# B&R Automation Studio project Panasonic_LinkaPowerCP2_A2021055 (part 40)

#### Main.st - Init, cyclic, exit code
```iecst
PROGRAM _INIT
	(* Insert code here *)

END_PROGRAM

PROGRAM _CYCLIC

	//Volanie funkcie SequenceControl//
    SequenceControl(SC:= SC_Devlink);

    //******************************************Štruktura nazvu adresára na serveri Panasonic************************************************//
    //Názov linky//
    StruktNovehoNazvuAdresara.LINKA:= 'PowerCP_CP4';

    //Názov pracoviska//
    StruktNovehoNazvuAdresara.PRACOVISKO:= 'ST10';

    //Rok//
    brsstrcpy(ADR(StruktNovehoNazvuAdresara.ROK),ADR(Rok_STR_4_Znaky));

    //Dátum//
    StruktNovehoNazvuAdresara.DATUM:= '';
    brsstrcat(ADR(StruktNovehoNazvuAdresara.DATUM),ADR(Rok_STR_4_Znaky));
    brsstrcat(ADR(StruktNovehoNazvuAdresara.DATUM),ADR('_'));
    brsstrcat(ADR(StruktNovehoNazvuAdresara.DATUM),ADR(Mesiac_STR));
    brsstrcat(ADR(StruktNovehoNazvuAdresara.DATUM),ADR('_'));
    brsstrcat(ADR(StruktNovehoNazvuAdresara.DATUM),ADR(Den_STR));

    //*********************************************Štruktura názvu premenovaného súboru v PLC***************************************************//
    //Datum//
    StruktNovehoNazvuSuboru.DATUM:= '';
    brsstrcat(ADR(StruktNovehoNazvuSuboru.DATUM),ADR(Rok_STR_4_Znaky));
    brsstrcat(ADR(StruktNovehoNazvuSuboru.DATUM),ADR('_'));
    brsstrcat(ADR(StruktNovehoNazvuSuboru.DATUM),ADR(Mesiac_STR));
    brsstrcat(ADR(StruktNovehoNazvuSuboru.DATUM),ADR('_'));
    brsstrcat(ADR(StruktNovehoNazvuSuboru.DATUM),ADR(Den_STR));

    //Čas//
    StruktNovehoNazvuSuboru.CAS:= '';
    brsstrcat(ADR(StruktNovehoNazvuSuboru.CAS),ADR(Hodina_STR));
    brsstrcat(ADR(StruktNovehoNazvuSuboru.CAS),ADR('_'));
    brsstrcat(ADR(StruktNovehoNazvuSuboru.CAS),ADR(Minuta_STR));
    brsstrcat(ADR(StruktNovehoNazvuSuboru.CAS),ADR('_'));
    brsstrcat(ADR(StruktNovehoNazvuSuboru.CAS),ADR(Sekunda_STR));

    //Kód modelu//
    StruktNovehoNazvuSuboru.SERIAL:= FTP_CAM16.INPUTS.QRkodPowerCP;

    //Index fotky//
    StruktNovehoNazvuSuboru.INDEX:= FTP_CAM16.INPUTS.IndexFotky;

    //Result fotky//
    StruktNovehoNazvuSuboru.RESULT:= FTP_CAM16.INPUTS.Result;

	//Prípona súboru//
	IF TypFotky_BMP THEN
		StruktNovehoNazvuSuboru.Pripona:= '.bmp';
	ELSE
		StruktNovehoNazvuSuboru.Pripona:= '.jpg';
	END_IF

    //Mapovanie premenných//
    FTP_CAM16.STATUS.AdresarPrazdny:= AdresarPrazdny;

	CASE SC_Devlink.Step OF

		0:
			SC_Devlink.StepName:= '0 - Nulovanie';
			FTP_CAM16.STATUS.KomunikaciaError:= FALSE;
			FTP_CAM16.STATUS.KomunikaciaUkoncena:= FALSE;
			PocetHladaniFotky:= 0;
            AdresarPrazdny:= FALSE;
            PocetNajdenychSuborov:= 0;
            PocetNajdenychAdresarov:= 0;
            PocetPremenovanychSuborov:= 0;
            PocetSkopirovanychSuborov:= 0;
            PocetVymazanychSuborov:= 0;
            i:= 0;
            PocetPokusov_FTP_KOM:= 0;
			PoruchaKomunikacie:= FALSE;
			DirInfo_0.enable:= FALSE;
			DirRead_0.enable:= FALSE;
			FileRename_0.enable:= FALSE;
			DirCreate_0.enable:= FALSE;
			DirInfo_0.enable:= FALSE;
			DirRead_0.enable:= FALSE;
			FileCopy_0.enable:= FALSE;
			FileDelete_0.enable:= FALSE;
			SC_Devlink.Step:= 1;

        1:
            SC_Devlink.StepName:= '1 - Rozhodnutie o cinnosti';
            IF FTP_CAM16.CMD.OdosliFotku THEN
                FTP_CAM16.STATUS.PopisPoruchy:= '';
                SC_Devlink.Step:= 15;
            ELSIF FTP_CAM16.CMD.VymazFotku THEN
                FTP_CAM16.STATUS.PopisPoruchy:= '';
                SC_Devlink.Step:= 153;
            END_IF

		15:
			SC_Devlink.StepName:= '15 - Odoslanie fotky, kontrola pripojenia na FTP server Panasonic';
			SC_Devlink.IdleTime.PT:= T#3s;
			SC_Devlink.AlarmTime.PT:= T#3s;

			IF Stav_PripojenieFTP_OK THEN
				SC_Devlink.ResetStep:= TRUE;
				SC_Devlink.Step:= 20;
			END_IF

        20:
            SC_Devlink.StepName:= '20 - Odoslanie fotky na server, nacitanie adresara kamery pred premenovanim';
            SC_Devlink.IdleTime.PT:= T#3s;
            SC_Devlink.AlarmTime.PT:= T#3s;

            DirInfo_0.enable:= TRUE;
            DirInfo_0.pDevice:= ADR('CAM16');
            DirInfo_0.pPath:= ADR('/');   //ak je nula tak číta všetky súbory a adresáre v koreni ak je "/Temp" tak číta všetky súbory a adresáre v adresári Temp//
            DirInfo_0();

            IF DirInfo_0.status = 0 THEN
                PocetNajdenychAdresarov:= DirInfo_0.dirnum;
                PocetNajdenychSuborov:= DirInfo_0.filenum;
                brsmemset(ADR(FileList[0]),0, SIZEOF(FileList));  //Vynulovanie pola stringov pre záznam adresárov a súborov
                SC_Devlink.ResetStep:= TRUE;
                SC_Devlink.Step:= 23;
            ELSIF DirInfo_0.status = 65535 THEN
                //BUSY//
            ELSIF DirInfo_0.status = 20723 THEN
                FTP_CAM16.STATUS.PopisPoruchy:= 'Porucha nacitania adresara kamery';
                Buffer_16.Hodnota:= DirInfo_0.status;
                Buffer_16.ZapisHodnotu:= TRUE;
                PoruchaKomunikacie:= TRUE;
                SC_Devlink.ResetStep:= TRUE;
                SC_Devlink.Step:= 100;
            ELSE
                FTP_CAM16.STATUS.PopisPoruchy:= 'Porucha nacitania adresara kamery';
                IF DirInfo_0.status = 20799 THEN
                    Buffer_16.Hodnota:= FileIoGetSysError();
                ELSE
                    Buffer_16.Hodnota:= DirInfo_0.status;
                END_IF
                Buffer_16.ZapisHodnotu:= TRUE;
                PoruchaKomunikacie:= TRUE;
                SC_Devlink.ResetStep:= TRUE;
                SC_Devlink.Step:= 100;
            END_IF

        23:
            SC_Devlink.StepName:= '23 - Odoslanie fotky na server, kontrola poctu najdenych suborov v adresari kamery';
            SC_Devlink.IdleTime.PT:= T#3s;
            SC_Devlink.AlarmTime.PT:= T#3s;

            IF PocetNajdenychSuborov > 0 THEN
                PocetHladaniFotky:= 0;
                SC_Devlink.ResetStep:= TRUE;
                SC_Devlink.Step:= 25;
            ELSIF PocetHladaniFotky < 100 THEN
                PocetHladaniFotky:= PocetHladaniFotky + 1;
                SC_Devlink.ResetStep:= TRUE;
                SC_Devlink.Step:= 20;
            ELSIF PocetHladaniFotky >= 100 THEN
                AdresarPrazdny:= TRUE;
                FTP_CAM16.STATUS.KomunikaciaUkoncena:= TRUE;
                SC_Devlink.ResetStep:= TRUE;
                SC_Devlink.Step:= 100;
            END_IF

        25:
            SC_Devlink.StepName:= '25 - Odoslanie fotky na server, zapis nazvou najdenych suborov do pola stringov';
            SC_Devlink.IdleTime.PT:= T#3s;
            SC_Devlink.AlarmTime.PT:= T#3s;

            DirRead_0.enable:= TRUE;
            DirRead_0.pDevice:= ADR('CAM16');
            DirRead_0.pPath:= ADR('/');   //ak je nula tak číta všetky súbory a adresáre v koreni ak je "/Temp" tak číta všetky súbory a adresáre v adresári Temp//
            DirRead_0.option:= fiFILE; //Zapíše súbory aj adresáre, ak je fiDIRECTORY zapíše len adresáre, ak je fiFILE tak zapíše len súbory//
            DirRead_0.entry:= i; //index zapisovania do pola//
            DirRead_0.pData:= ADR(ReadData);
            DirRead_0.data_len:= SIZEOF(ReadData);
            DirRead_0();

            IF DirRead_0.status = 0 THEN
                brsstrcpy(ADR(FileList[i]), ADR(ReadData.Filename[0])); //Uloženie názvou adresárov a súborov do pola stringov
				IF i< 100 THEN
					i:= i + 1;
				END_IF
            ELSIF DirRead_0.status = 20702 THEN
                i:= 0;
                SC_Devlink.ResetStep:= TRUE;
                SC_Devlink.Step:= 28;
            ELSIF DirRead_0.status = 65535 THEN
                //BUSY//
            ELSE
                FTP_CAM16.STATUS.PopisPoruchy:= 'Porucha zapisu suborov do pola';
                PoruchaKomunikacie:= TRUE;
                SC_Devlink.ResetStep:= TRUE;
                SC_Devlink.Step:= 100;
            END_IF

        28:
            SC_Devlink.StepName:= '28 - Odoslanie fotky na server, premenovanie fotky';
            SC_Devlink.IdleTime.PT:= T#3s;
            SC_Devlink.AlarmTime.PT:= T#3s;

            StaryNazovSuboru:= '';
            brsstrcat(ADR(StaryNazovSuboru),ADR('/'));
            brsstrcat(ADR(StaryNazovSuboru),ADR(FileList[i]));

            NovyNazovSuboru:= '';
            brsstrcat(ADR(NovyNazovSuboru),ADR('/'));
            brsstrcat(ADR(NovyNazovSuboru),ADR(StruktNovehoNazvuSuboru.DATUM));
            brsstrcat(ADR(NovyNazovSuboru),ADR('_'));
            brsstrcat(ADR(NovyNazovSuboru),ADR(StruktNovehoNazvuSuboru.CAS));
            brsstrcat(ADR(NovyNazovSuboru),ADR('_'));
            brsstrcat(ADR(NovyNazovSuboru),ADR(StruktNovehoNazvuSuboru.SERIAL));
            brsstrcat(ADR(NovyNazovSuboru),ADR('_'));
            brsstrcat(ADR(NovyNazovSuboru),ADR(StruktNovehoNazvuSuboru.INDEX));
            brsstrcat(ADR(NovyNazovSuboru),ADR('_'));
            brsstrcat(ADR(NovyNazovSuboru),ADR(StruktNovehoNazvuSuboru.RESULT));
            brsstrcat(ADR(NovyNazovSuboru),ADR(StruktNovehoNazvuSuboru.Pripona));

            FileRename_0.enable:= TRUE;
            FileRename_0.pDevice:= ADR('CAM16');
            FileRename_0.pName:= ADR(StaryNazovSuboru);
            FileRename_0.pNewName:= ADR(NovyNazovSuboru);
            FileRename_0();

            IF FileRename_0.status = 0 THEN
                SC_Devlink.ResetStep:= TRUE;
                SC_Devlink.Step:= 30;
            ELSIF FileRename_0.status = 65535 THEN
                //BUSY//
            ELSIF FileRename_0.status = 20705 THEN
                SC_Devlink.ResetStep:= TRUE;
                SC_Devlink.Step:= 30;
            ELSIF FileRename_0.status = 20708 THEN
                AdresarPrazdny:= TRUE;
                FTP_CAM16.STATUS.KomunikaciaUkoncena:= TRUE;
                SC_Devlink.ResetStep:= TRUE;
                SC_Devlink.Step:= 100;
            ELSE
                FTP_CAM16.STATUS.PopisPoruchy:= 'Porucha premenovania fotky';
				PoruchaKomunikacie:= TRUE;
                SC_Devlink.ResetStep:= TRUE;
                SC_Devlink.Step:= 100;
            END_IF

        30:
            SC_Devlink.StepName:= '30 - Odoslanie fotky na server, kontrola poctu premenovanych suborov';
            SC_Devlink.IdleTime.PT:= T#3s;
            SC_Devlink.AlarmTime.PT:= T#3s;

            IF NOT SC_Devlink.Switch1 THEN
                PocetPremenovanychSuborov:= PocetPremenovanychSuborov + 1;
                SC_Devlink.Switch1:= TRUE;
            END_IF

            IF PocetPremenovanychSuborov < PocetNajdenychSuborov THEN
                IF i< 100 THEN
					i:= i + 1;
				END_IF
                SC_Devlink.ResetStep:= TRUE;
                SC_Devlink.Step:= 28;
            ELSE
                i:= 0;
                PocetNajdenychSuborov:= 0;
                PocetNajdenychAdresarov:= 0;
                SC_Devlink.ResetStep:= TRUE;
                SC_Devlink.Step:= 33;//33
            END_IF

        33: SC_Devlink.StepName:= '33 - Odoslanie fotky na server, vytvorenie adresara LINKA';
            SC_Devlink.IdleTime.PT:= T#3s;
            SC_Devlink.AlarmTime.PT:= T#3s;

            NazovAdresara_LINKA:= '';
            brsstrcat(ADR(NazovAdresara_LINKA),ADR('DesignMP'));
            brsstrcat(ADR(NazovAdresara_LINKA),ADR('/'));
            brsstrcat(ADR(NazovAdresara_LINKA),ADR(StruktNovehoNazvuAdresara.LINKA));

            DirCreate_0.enable:= TRUE;
            DirCreate_0.pDevice:= ADR('Panasonic');
            DirCreate_0.pName:= ADR(NazovAdresara_LINKA);
            DirCreate_0();

            IF DirCreate_0.status = 0 THEN
                SC_Devlink.ResetStep:= TRUE;
                SC_Devlink.Step:= 35;
            ELSIF DirCreate_0.status = 65535 THEN
                //BUSY//
            ELSIF DirCreate_0.status = 20725 THEN
                SC_Devlink.ResetStep:= TRUE;
                SC_Devlink.Step:= 35;
            ELSIF DirCreate_0.status = 20709 THEN
                //BUSY//
            ELSE
                FTP_CAM16.STATUS.PopisPoruchy:= 'Porucha vytvorenia adresara na FTP Panasonic';
                PoruchaKomunikacie:= TRUE;
                SC_Devlink.ResetStep:= TRUE;
                SC_Devlink.Step:= 100;
            END_IF

        35: SC_Devlink.StepName:= '35 - Odoslanie fotky na server, vytvorenie podadresara PRACOVISKO';
            SC_Devlink.IdleTime.PT:= T#3s;
            SC_Devlink.AlarmTime.PT:= T#3s;

            NazovPodAdresara_PRACOVISKO:= '';
            brsstrcat(ADR(NazovPodAdresara_PRACOVISKO),ADR(NazovAdresara_LINKA));
            brsstrcat(ADR(NazovPodAdresara_PRACOVISKO),ADR('/'));
            brsstrcat(ADR(NazovPodAdresara_PRACOVISKO),ADR(StruktNovehoNazvuAdresara.PRACOVISKO));

            DirCreate_0.enable:= TRUE;
            DirCreate_0.pDevice:= ADR('Panasonic');
            DirCreate_0.pName:= ADR(NazovPodAdresara_PRACOVISKO);
            DirCreate_0();

            IF DirCreate_0.status = 0 THEN
                SC_Devlink.ResetStep:= TRUE;
                SC_Devlink.Step:= 38;
            ELSIF DirCreate_0.status = 65535 THEN
                //BUSY//
            ELSIF DirCreate_0.status = 20725 THEN
                SC_Devlink.ResetStep:= TRUE;
                SC_Devlink.Step:= 38;
            ELSIF DirCreate_0.status = 20709 THEN
                //BUSY//
            ELSE
                FTP_CAM16.STATUS.PopisPoruchy:= 'Porucha vytvorenia adresara na FTP Panasonic';
                PoruchaKomunikacie:= TRUE;
                SC_Devlink.ResetStep:= TRUE;
                SC_Devlink.Step:= 100;
            END_IF

        38: SC_Devlink.StepName:= '38 - Odoslanie fotky na server, vytvorenie podadresara ROK';
            SC_Devlink.IdleTime.PT:= T#3s;
            SC_Devlink.AlarmTime.PT:= T#3s;

            NazovPodAdresara_ROK:= '';
            brsstrcat(ADR(NazovPodAdresara_ROK),ADR(NazovPodAdresara_PRACOVISKO));
            brsstrcat(ADR(NazovPodAdresara_ROK),ADR('/'));
            brsstrcat(ADR(NazovPodAdresara_ROK),ADR(StruktNovehoNazvuAdresara.ROK));

            DirCreate_0.enable:= TRUE;
            DirCreate_0.pDevice:= ADR('Panasonic');
            DirCreate_0.pName:= ADR(NazovPodAdresara_ROK);
            DirCreate_0();

            IF DirCreate_0.status = 0 THEN
                SC_Devlink.ResetStep:= TRUE;
                SC_Devlink.Step:= 40;
            ELSIF DirCreate_0.status = 65535 THEN
                //BUSY//
            ELSIF DirCreate_0.status = 20725 THEN
                SC_Devlink.ResetStep:= TRUE;
                SC_Devlink.Step:= 40;
            ELSIF DirCreate_0.status = 20709 THEN
                //BUSY//
            ELSE
                FTP_CAM16.STATUS.PopisPoruchy:= 'Porucha vytvorenia adresara na FTP Panasonic';
                PoruchaKomunikacie:= TRUE;
                SC_Devlink.ResetStep:= TRUE;
                SC_Devlink.Step:= 100;
            END_IF

        40: SC_Devlink.StepName:= '40 - Odoslanie fotky na server, vytvorenie podadresara DATUM';
            SC_Devlink.IdleTime.PT:= T#3s;
            SC_Devlink.AlarmTime.PT:= T#3s;

            NazovPodAdresara_DATUM:= '';
            brsstrcat(ADR(NazovPodAdresara_DATUM),ADR(NazovPodAdresara_ROK));
            brsstrcat(ADR(NazovPodAdresara_DATUM),ADR('/'));
            brsstrcat(ADR(NazovPodAdresara_DATUM),ADR(StruktNovehoNazvuAdresara.DATUM));

            DirCreate_0.enable:= TRUE;
            DirCreate_0.pDevice:= ADR('Panasonic');
            DirCreate_0.pName:= ADR(NazovPodAdresara_DATUM);
            DirCreate_0();

            IF DirCreate_0.status = 0 THEN
                SC_Devlink.ResetStep:= TRUE;
                SC_Devlink.Step:= 43;
            ELSIF DirCreate_0.status = 65535 THEN
                //BUSY//
            ELSIF DirCreate_0.status = 20725 THEN
                SC_Devlink.ResetStep:= TRUE;
                SC_Devlink.Step:= 43;
            ELSIF DirCreate_0.status = 20709 THEN
                //BUSY//
            ELSE
                FTP_CAM16.STATUS.PopisPoruchy:= 'Porucha vytvorenia adresara na FTP Panasonic';
                PoruchaKomunikacie:= TRUE;
                SC_Devlink.ResetStep:= TRUE;
                SC_Devlink.Step:= 100;
            END_IF

        43:	SC_Devlink.StepName:= '43 - Odoslanie fotky na server, nacitanie adresara pred kopirovanim fotiek na server Panasonic';
            SC_Devlink.IdleTime.PT:= T#3s;
            SC_Devlink.AlarmTime.PT:= T#3s;

            DirInfo_0.enable:= TRUE;
            DirInfo_0.pDevice:= ADR('CAM16');
            DirInfo_0.pPath:= ADR('/');   //ak je nula tak číta všetky súbory a adresáre v koreni ak je "/Temp" tak číta všetky súbory a adresáre v adresári Temp//
            DirInfo_0();

            IF DirInfo_0.status = 0 THEN
                PocetNajdenychAdresarov:= DirInfo_0.dirnum;
                PocetNajdenychSuborov:= DirInfo_0.filenum;
                brsmemset(ADR(FileList[0]),0, SIZEOF(FileList));  //Vynulovanie pola stringov pre záznam adresárov a súborov
                SC_Devlink.ResetStep:= TRUE;
                SC_Devlink.Step:= 45;
            ELSIF DirInfo_0.status = 65535 THEN
                //BUSY//
            ELSIF DirInfo_0.status = 20723 THEN
                FTP_CAM16.STATUS.PopisPoruchy:= 'Porucha nacitania adresara kamery';
                Buffer_16.Hodnota:= DirInfo_0.status;
                Buffer_16.ZapisHodnotu:= TRUE;
                PoruchaKomunikacie:= TRUE;
                SC_Devlink.ResetStep:= TRUE;
                SC_Devlink.Step:= 100;
            ELSE
                FTP_CAM16.STATUS.PopisPoruchy:= 'Porucha nacitania adresara kamery';
                IF DirInfo_0.status = 20799 THEN
                    Buffer_16.Hodnota:= FileIoGetSysError();
                ELSE
                    Buffer_16.Hodnota:= DirInfo_0.status;
                END_IF
                Buffer_16.ZapisHodnotu:= TRUE;
                PoruchaKomunikacie:= TRUE;
                SC_Devlink.ResetStep:= TRUE;
                SC_Devlink.Step:= 100;
            END_IF

        45: SC_Devlink.StepName:= '45 - Odoslanie fotky na server, zapis nazvou najdenych suborov do pola stringov';
            SC_Devlink.IdleTime.PT:= T#3s;
            SC_Devlink.AlarmTime.PT:= T#3s;

            DirRead_0.enable:= TRUE;
            DirRead_0.pDevice:= ADR('CAM16');
            DirRead_0.pPath:= ADR('/');   //ak je nula tak číta všetky súbory a adresáre v koreni ak je "/Temp" tak číta všetky súbory a adresáre v adresári Temp//
            DirRead_0.option:= fiFILE; //Zapíše súbory aj adresáre, ak je fiDIRECTORY zapíše len adresáre, ak je fiFILE tak zapíše len súbory//
            DirRead_0.entry:= i; //index zapisovania do pola//
            DirRead_0.pData:= ADR(ReadData);
            DirRead_0.data_len:= SIZEOF(ReadData);
            DirRead_0();

            IF DirRead_0.status = 0 THEN
                brsstrcpy(ADR(FileList[i]), ADR(ReadData.Filename[0])); //Uloženie názvou adresárov a súborov do pola stringov
				IF i< 100 THEN
					i:= i + 1;
				END_IF
            ELSIF DirRead_0.status = 20702 THEN
                i:= 0;
                SC_Devlink.ResetStep:= TRUE;
                SC_Devlink.Step:= 47;
            ELSIF DirRead_0.status = 65535 THEN
                //BUSY//
            ELSE
                FTP_CAM16.STATUS.PopisPoruchy:= 'Porucha zapisu najdenych suborov do pola';
                PoruchaKomunikacie:= TRUE;
                SC_Devlink.ResetStep:= TRUE;
                SC_Devlink.Step:= 100;
            END_IF

		47:
			SC_Devlink.StepName:= '47 - Odoslanie fotky na server, vytvorenie cesty pre kopírovanie suboruk fotky na server Panasonic';
			SC_Devlink.IdleTime.PT:= T#3s;
			SC_Devlink.AlarmTime.PT:= T#3s;

			ZdrojKopirovaniaSuboru:= '';
			brsstrcat(ADR(ZdrojKopirovaniaSuboru),ADR('/'));
			brsstrcat(ADR(ZdrojKopirovaniaSuboru),ADR(ReadData.Filename));

			CielKopirovaniaSuboru:= '';
			brsstrcat(ADR(CielKopirovaniaSuboru),ADR(NazovPodAdresara_DATUM));
			brsstrcat(ADR(CielKopirovaniaSuboru),ADR('/'));
			brsstrcat(ADR(CielKopirovaniaSuboru),ADR(ReadData.Filename));

			SC_Devlink.ResetStep:= TRUE;
			SC_Devlink.Step:= 48;

        48: SC_Devlink.StepName:= '48 - Odoslanie fotky na server, kopirovanie fotky na server Panasonic';
            SC_Devlink.IdleTime.PT:= T#3s;
            SC_Devlink.AlarmTime.PT:= T#3s;

			FileCopy_0.enable:= TRUE;
			FileCopy_0.pSrcDev:= ADR('CAM16'); //Zdrojové zariadenie od kial sa kopíruje
			FileCopy_0.pSrc:= ADR(ZdrojKopirovaniaSuboru);
			FileCopy_0.pDestDev:= ADR('Panasonic'); //Cielové zariadenie kam sa má súbor skopírovať
			FileCopy_0.pDest:= ADR(CielKopirovaniaSuboru);
			FileCopy_0.option := fiOVERWRITE;
			FileCopy_0();

            IF FileCopy_0.status = 0 THEN
                SC_Devlink.ResetStep:= TRUE;
                SC_Devlink.Step:= 50;
            ELSIF FileCopy_0.status = 65535 THEN
                //BUSY//
            ELSIF FileCopy_0.status = 20705 THEN
                SC_Devlink.ResetStep:= TRUE;
				SC_Devlink.Step:= 50;
			ELSIF FileCopy_0.status = 20799 THEN
				SC_Devlink.ResetStep:= TRUE;
				SC_Devlink.Step:= 50;
            ELSIF FileCopy_0.status = 20708 THEN
                AdresarPrazdny:= TRUE;
                FTP_CAM16.STATUS.KomunikaciaUkoncena:= TRUE;
                SC_Devlink.ResetStep:= TRUE;
                SC_Devlink.Step:= 100;
            ELSE
                FTP_CAM16.STATUS.PopisPoruchy:= 'Porucha kopirovania fotky na FTP Panasonic';
                PoruchaKomunikacie:= TRUE;
                SC_Devlink.ResetStep:= TRUE;
                SC_Devlink.Step:= 100;
            END_IF

        50: SC_Devlink.StepName:= '50 - Odoslanie fotky na server, kontrola poctu skopirovanych suborov';
            SC_Devlink.IdleTime.PT:= T#3s;
            SC_Devlink.AlarmTime.PT:= T#3s;

            IF NOT SC_Devlink.Switch1 THEN
                PocetSkopirovanychSuborov:= PocetSkopirovanychSuborov + 1;
                SC_Devlink.Switch1:= TRUE;
            END_IF

            IF PocetSkopirovanychSuborov < PocetNajdenychSuborov THEN
                IF i< 100 THEN
					i:= i + 1;
				END_IF
                SC_Devlink.ResetStep:= TRUE;
                SC_Devlink.Step:= 48;
            ELSE
                i:= 0;
                PocetNajdenychSuborov:= 0;
                PocetNajdenychAdresarov:= 0;
                SC_Devlink.ResetStep:= TRUE;
                SC_Devlink.Step:= 60;
            END_IF

        60:
            SC_Devlink.StepName:= '60 - Odoslanie fotky na server, nacitanie adresara kamery pred vymazanim';
            SC_Devlink.IdleTime.PT:= T#3s;
            SC_Devlink.AlarmTime.PT:= T#3s;

            DirInfo_0.enable:= TRUE;
            DirInfo_0.pDevice:= ADR('CAM16');
            DirInfo_0.pPath:= ADR('/');   //ak je nula tak číta všetky súbory a adresáre v koreni ak je "/Temp" tak číta všetky súbory a adresáre v adresári Temp//
            DirInfo_0();

            IF DirInfo_0.status = 0 THEN
                PocetNajdenychAdresarov:= DirInfo_0.dirnum;
                PocetNajdenychSuborov:= DirInfo_0.filenum;
                brsmemset(ADR(FileList[0]),0, SIZEOF(FileList));  //Vynulovanie pola stringov pre záznam adresárov a súborov
                SC_Devlink.Step:= 63;
            ELSIF DirInfo_0.status = 65535 THEN
                //BUSY//
            ELSIF DirInfo_0.status = 20723 THEN
                FTP_CAM16.STATUS.PopisPoruchy:= 'Porucha nacitania adresara kamery';
                Buffer_16.Hodnota:= DirInfo_0.status;
                Buffer_16.ZapisHodnotu:= TRUE;
                PoruchaKomunikacie:= TRUE;
                SC_Devlink.ResetStep:= TRUE;
                SC_Devlink.Step:= 100;
            ELSE
                FTP_CAM16.STATUS.PopisPoruchy:= 'Porucha nacitania adresara kamery';
                IF DirInfo_0.status = 20799 THEN
                    Buffer_16.Hodnota:= FileIoGetSysError();
                ELSE
                    Buffer_16.Hodnota:= DirInfo_0.status;
                END_IF
                Buffer_16.ZapisHodnotu:= TRUE;
                PoruchaKomunikacie:= TRUE;
                SC_Devlink.ResetStep:= TRUE;
                SC_Devlink.Step:= 100;
            END_IF

        63: SC_Devlink.StepName:= '63 - Odoslanie fotky na server, zapis nazvou najdenych suborov do pola stringov';
            SC_Devlink.IdleTime.PT:= T#3s;
            SC_Devlink.AlarmTime.PT:= T#3s;

            DirRead_0.enable:= TRUE;
            DirRead_0.pDevice:= ADR('CAM16');
            DirRead_0.pPath:= ADR('/');   //ak je nula tak číta všetky súbory a adresáre v koreni ak je "/Temp" tak číta všetky súbory a adresáre v adresári Temp//
            DirRead_0.option:= fiFILE; //Zapíše súbory aj adresáre, ak je fiDIRECTORY zapíše len adresáre, ak je fiFILE tak zapíše len súbory//
            DirRead_0.entry:= i; //index zapisovania do pola//
            DirRead_0.pData:= ADR(ReadData);
            DirRead_0.data_len:= SIZEOF(ReadData);
            DirRead_0();

            IF DirRead_0.status = 0 THEN
                brsstrcpy(ADR(FileList[i]), ADR(ReadData.Filename[0])); //Uloženie názvou adresárov a súborov do pola stringov
				IF i< 100 THEN
					i:= i + 1;
				END_IF
            ELSIF DirRead_0.status = 20702 THEN
                i:= 0;
                SC_Devlink.ResetStep:= TRUE;
                SC_Devlink.Step:= 65;
            ELSIF DirRead_0.status = 65535 THEN
                //BUSY//
            ELSE
                FTP_CAM16.STATUS.PopisPoruchy:= 'Porucha zapisu najdenych suborov do pola';
                PoruchaKomunikacie:= TRUE;
                SC_Devlink.ResetStep:= TRUE;
                SC_Devlink.Step:= 100;
            END_IF

        65: SC_Devlink.StepName:= '65 - Odoslanie fotky na server, vymazanie suboru';
            SC_Devlink.IdleTime.PT:= T#3s;
            SC_Devlink.AlarmTime.PT:= T#3s;

            ZdrojKopirovaniaSuboru:= '';
            brsstrcat(ADR(ZdrojKopirovaniaSuboru),ADR('/'));
            brsstrcat(ADR(ZdrojKopirovaniaSuboru),ADR(FileList[i]));

            FileDelete_0.enable:= TRUE;
            FileDelete_0.pDevice:= ADR('CAM16');
            FileDelete_0.pName:= ADR(ZdrojKopirovaniaSuboru);
            FileDelete_0();

            IF FileDelete_0.status = 0 THEN
                SC_Devlink.ResetStep:= TRUE;
                SC_Devlink.Step:= 68;
            ELSIF FileDelete_0.status = 65535 THEN
                //BUSY//
            ELSIF FileDelete_0.status = 20708 THEN
                SC_Devlink.ResetStep:= TRUE;
                SC_Devlink.Step:= 68;
            ELSE
                FTP_CAM16.STATUS.PopisPoruchy:= 'Porucha vymazania fotky v adresari kamery';
                PoruchaKomunikacie:= TRUE;
                SC_Devlink.ResetStep:= TRUE;
                SC_Devlink.Step:= 100;
            END_IF

        68:	SC_Devlink.StepName:= '68 - Odoslanie fotky na server, kontrola poctu vymazanych suborov';
            SC_Devlink.IdleTime.PT:= T#3s;
            SC_Devlink.AlarmTime.PT:= T#3s;

            IF NOT SC_Devlink.Switch1 THEN
                PocetVymazanychSuborov:= PocetVymazanychSuborov + 1;
                SC_Devlink.Switch1:= TRUE;
            END_IF

            IF PocetVymazanychSuborov < PocetNajdenychSuborov THEN
                IF i< 100 THEN
					i:= i + 1;
				END_IF
                SC_Devlink.ResetStep:= TRUE;
                SC_Devlink.Step:= 65;
            ELSE
                i:= 0;
                PocetNajdenychSuborov:= 0;
                PocetNajdenychAdresarov:= 0;
                CAM16_PocetFotiek:= 0;
				FTP_CAM16.STATUS.KomunikaciaUkoncena:= TRUE;
                SC_Devlink.ResetStep:= TRUE;
                SC_Devlink.Step:= 100;
            END_IF

        100:
            SC_Devlink.StepName:= '100 - Odoslanie fotky, cakam na zrusenie prikazu odosli fotku';
            SC_Devlink.IdleTime.PT:= T#1s;
            SC_Devlink.AlarmTime.PT:= T#3s;

            SC_Devlink.IdleTime.IN:= TRUE;

            IF PoruchaKomunikacie AND SC_Devlink.IdleTime.Q AND PocetPokusov_FTP_KOM < 3 THEN
                PocetPokusov_FTP_KOM:= PocetPokusov_FTP_KOM + 1;
                PoruchaKomunikacie:= FALSE;
                i:= 0;
                PocetNajdenychSuborov:= 0;
                PocetNajdenychAdresarov:= 0;
                SC_Devlink.ResetStep:= TRUE;
                SC_Devlink.Step:= 1;
            ELSIF PoruchaKomunikacie AND PocetPokusov_FTP_KOM >= 3 THEN
                FTP_CAM16.STATUS.KomunikaciaError:= TRUE;
            END_IF

            IF NOT FTP_CAM16.CMD.OdosliFotku THEN
                SC_Devlink.ResetStep:= TRUE;
                SC_Devlink.Step:= 0;
            END_IF

            //**************************************Vymazanie fotky*************************************************//

		153:
			SC_Devlink.StepName:= '153 - Vymazanie fotky, nacitanie adresara kamery pred vymazanim';
			SC_Devlink.IdleTime.PT:= T#3s;
			SC_Devlink.AlarmTime.PT:= T#3s;

			DirInfo_0.enable:= TRUE;
			DirInfo_0.pDevice:= ADR('CAM16');
			DirInfo_0.pPath:= ADR('/');   //ak je nula tak číta všetky súbory a adresáre v koreni ak je "/Temp" tak číta všetky súbory a adresáre v adresári Temp//
			DirInfo_0();

			IF DirInfo_0.status = 0 THEN
				PocetNajdenychAdresarov:= DirInfo_0.dirnum;
				PocetNajdenychSuborov:= DirInfo_0.filenum;
				brsmemset(ADR(FileList[0]),0, SIZEOF(FileList));  //Vynulovanie pola stringov pre záznam adresárov a súborov
				SC_Devlink.Step:= 155;
			ELSIF DirInfo_0.status = 65535 THEN
				//BUSY//
			ELSIF DirInfo_0.status = 20723 THEN
				FTP_CAM16.STATUS.PopisPoruchy:= 'Porucha nacitania adresara kamery';
				Buffer_16.Hodnota:= DirInfo_0.status;
				Buffer_16.ZapisHodnotu:= TRUE;
				PoruchaKomunikacie:= TRUE;
				SC_Devlink.ResetStep:= TRUE;
				SC_Devlink.Step:= 200;
			ELSE
				FTP_CAM16.STATUS.PopisPoruchy:= 'Porucha nacitania adresara kamery';
				IF DirInfo_0.status = 20799 THEN
					Buffer_16.Hodnota:= FileIoGetSysError();
				ELSE
					Buffer_16.Hodnota:= DirInfo_0.status;
				END_IF
				Buffer_16.ZapisHodnotu:= TRUE;
				PoruchaKomunikacie:= TRUE;
				SC_Devlink.ResetStep:= TRUE;
				SC_Devlink.Step:= 200;
			END_IF

		155: SC_Devlink.StepName:= '155 - Vymazanie fotky, zapis nazvou najdenych suborov do pola stringov';
			SC_Devlink.IdleTime.PT:= T#3s;
			SC_Devlink.AlarmTime.PT:= T#3s;

			DirRead_0.enable:= TRUE;
			DirRead_0.pDevice:= ADR('CAM16');
			DirRead_0.pPath:= ADR('/');   //ak je nula tak číta všetky súbory a adresáre v koreni ak je "/Temp" tak číta všetky súbory a adresáre v adresári Temp//
			DirRead_0.option:= fiFILE; //Zapíše súbory aj adresáre, ak je fiDIRECTORY zapíše len adresáre, ak je fiFILE tak zapíše len súbory//
			DirRead_0.entry:= i; //index zapisovania do pola//
			DirRead_0.pData:= ADR(ReadData);
			DirRead_0.data_len:= SIZEOF(ReadData);
			DirRead_0();

			IF DirRead_0.status = 0 THEN
				brsstrcpy(ADR(FileList[i]), ADR(ReadData.Filename[0])); //Uloženie názvou adresárov a súborov do pola stringov
				IF i< 100 THEN
					i:= i + 1;
				END_IF
			ELSIF DirRead_0.status = 20702 THEN
				i:= 0;
				SC_Devlink.ResetStep:= TRUE;
				SC_Devlink.Step:= 158;
			ELSIF DirRead_0.status = 65535 THEN
				//BUSY//
			ELSE
				FTP_CAM16.STATUS.PopisPoruchy:= 'Porucha zapisu najdenych suborov do pola';
				PoruchaKomunikacie:= TRUE;
				SC_Devlink.ResetStep:= TRUE;
				SC_Devlink.Step:= 200;
			END_IF

		158: SC_Devlink.StepName:= '158 - Vymazanie fotky, vymazanie suboru';
			SC_Devlink.IdleTime.PT:= T#3s;
			SC_Devlink.AlarmTime.PT:= T#3s;

			ZdrojKopirovaniaSuboru:= '';
			brsstrcat(ADR(ZdrojKopirovaniaSuboru),ADR('/'));
			brsstrcat(ADR(ZdrojKopirovaniaSuboru),ADR(FileList[i]));

			FileDelete_0.enable:= TRUE;
			FileDelete_0.pDevice:= ADR('CAM16');
			FileDelete_0.pName:= ADR(ZdrojKopirovaniaSuboru);
			FileDelete_0();

			IF FileDelete_0.status = 0 THEN
				SC_Devlink.ResetStep:= TRUE;
				SC_Devlink.Step:= 160;
            ELSIF FileDelete_0.status = 65535 THEN
                //BUSY//
            ELSIF FileDelete_0.status = 20708 THEN
                SC_Devlink.ResetStep:= TRUE;
                SC_Devlink.Step:= 160;
            ELSE
                FTP_CAM16.STATUS.PopisPoruchy:= 'Porucha vymazania fotky v adresari kamery';
                PoruchaKomunikacie:= TRUE;
                SC_Devlink.ResetStep:= TRUE;
                SC_Devlink.Step:= 200;
            END_IF

        160:	SC_Devlink.StepName:= '160 - Vymazanie fotky, kontrola poctu vymazanych suborov';
            SC_Devlink.IdleTime.PT:= T#3s;
            SC_Devlink.AlarmTime.PT:= T#3s;

            IF NOT SC_Devlink.Switch1 THEN
                PocetVymazanychSuborov:= PocetVymazanychSuborov + 1;
                SC_Devlink.Switch1:= TRUE;
            END_IF

            IF PocetVymazanychSuborov < PocetNajdenychSuborov THEN
                IF i< 100 THEN
					i:= i + 1;
				END_IF
                SC_Devlink.ResetStep:= TRUE;
                SC_Devlink.Step:= 158;
            ELSE
                i:= 0;
                PocetNajdenychSuborov:= 0;
                PocetNajdenychAdresarov:= 0;
                CAM16_PocetFotiek:= 0;
				FTP_CAM16.STATUS.KomunikaciaUkoncena:= TRUE;
                SC_Devlink.ResetStep:= TRUE;
                SC_Devlink.Step:= 200;
            END_IF

        200:
            SC_Devlink.StepName:= '200 - Vymazanie fotky, cakam na zrusenie prikazu odosli fotku';
            SC_Devlink.IdleTime.PT:= T#1s;
            SC_Devlink.AlarmTime.PT:= T#3s;

            SC_Devlink.IdleTime.IN:= TRUE;

            IF PoruchaKomunikacie AND SC_Devlink.IdleTime.Q AND PocetPokusov_FTP_KOM < 3 THEN
                PocetPokusov_FTP_KOM:= PocetPokusov_FTP_KOM + 1;
                PoruchaKomunikacie:= FALSE;
                i:= 0;
                PocetNajdenychSuborov:= 0;
                PocetNajdenychAdresarov:= 0;
                SC_Devlink.ResetStep:= TRUE;
                SC_Devlink.Step:= 1;
            ELSIF PoruchaKomunikacie AND PocetPokusov_FTP_KOM >= 3 THEN
                FTP_CAM16.STATUS.KomunikaciaError:= TRUE;
            END_IF

            IF NOT FTP_CAM16.CMD.VymazFotku THEN
                SC_Devlink.ResetStep:= TRUE;
                SC_Devlink.Step:= 0;
            END_IF

    END_CASE

END_PROGRAM

PROGRAM _EXIT
	(* Insert code here *)

END_PROGRAM
```

#### Variables.var - Local variables
```iecst
VAR
	SC_Devlink : SequenceControlTyp;
	DirInfo_0 : DirInfo;
	DirRead_0 : DirRead;
	FileRename_0 : FileRename;
	FileDelete_0 : FileDelete;
	FileCopy_0 : FileCopy;
	DirCreate_0 : DirCreate;
	i : UDINT;
	FileList : ARRAY[0..100] OF STRING[100];
	ReadData : fiDIR_READ_DATA; (*data-structure for command bDirRead*)
	PocetNajdenychAdresarov : UDINT;
	PocetNajdenychSuborov : UDINT;
	PocetPremenovanychSuborov : UDINT;
	PocetSkopirovanychSuborov : UDINT;
	PocetVymazanychSuborov : UDINT;
	StaryNazovSuboru : STRING[200];
	NovyNazovSuboru : STRING[200];
	ZdrojKopirovaniaSuboru : STRING[200];
	CielKopirovaniaSuboru : STRING[200];
	AdresarPrazdny : BOOL;
	StruktNovehoNazvuSuboru : StrukturaNovehoNazvuSuboru_typ;
	StruktNovehoNazvuAdresara : StrukturaNovehoNazvuAdresara_typ;
	NazovAdresara_LINKA : STRING[50];
	NazovPodAdresara_PRACOVISKO : STRING[50];
	NazovPodAdresara_ROK : STRING[50];
	NazovPodAdresara_DATUM : STRING[50];
	PocetHladaniFotky : UDINT;
	PocetPokusov_FTP_KOM : USINT;
	PoruchaKomunikacie : BOOL;
END_VAR
```

### Program Logical/OdosielanieFotiek/FTP_CAM17 (IEC)

#### Main.st - Init, cyclic, exit code
```iecst
PROGRAM _INIT
	(* Insert code here *)

END_PROGRAM

PROGRAM _CYCLIC

    //Volanie funkcie SequenceControl//
    SequenceControl(SC:= SC_Devlink);

    //******************************************Štruktura nazvu adresára na serveri Panasonic************************************************//
    //Názov linky//
    StruktNovehoNazvuAdresara.LINKA:= 'PowerCP_CP4';

    //Názov pracoviska//
    StruktNovehoNazvuAdresara.PRACOVISKO:= 'ST3';

    //Rok//
    brsstrcpy(ADR(StruktNovehoNazvuAdresara.ROK),ADR(Rok_STR_4_Znaky));

    //Dátum//
    StruktNovehoNazvuAdresara.DATUM:= '';
    brsstrcat(ADR(StruktNovehoNazvuAdresara.DATUM),ADR(Rok_STR_4_Znaky));
    brsstrcat(ADR(StruktNovehoNazvuAdresara.DATUM),ADR('_'));
    brsstrcat(ADR(StruktNovehoNazvuAdresara.DATUM),ADR(Mesiac_STR));
    brsstrcat(ADR(StruktNovehoNazvuAdresara.DATUM),ADR('_'));
    brsstrcat(ADR(StruktNovehoNazvuAdresara.DATUM),ADR(Den_STR));

    //*********************************************Štruktura názvu premenovaného súboru v PLC***************************************************//
    //Datum//
    StruktNovehoNazvuSuboru.DATUM:= '';
    brsstrcat(ADR(StruktNovehoNazvuSuboru.DATUM),ADR(Rok_STR_4_Znaky));
    brsstrcat(ADR(StruktNovehoNazvuSuboru.DATUM),ADR('_'));
    brsstrcat(ADR(StruktNovehoNazvuSuboru.DATUM),ADR(Mesiac_STR));
    brsstrcat(ADR(StruktNovehoNazvuSuboru.DATUM),ADR('_'));
    brsstrcat(ADR(StruktNovehoNazvuSuboru.DATUM),ADR(Den_STR));

    //Čas//
    StruktNovehoNazvuSuboru.CAS:= '';
    brsstrcat(ADR(StruktNovehoNazvuSuboru.CAS),ADR(Hodina_STR));
    brsstrcat(ADR(StruktNovehoNazvuSuboru.CAS),ADR('_'));
    brsstrcat(ADR(StruktNovehoNazvuSuboru.CAS),ADR(Minuta_STR));
    brsstrcat(ADR(StruktNovehoNazvuSuboru.CAS),ADR('_'));
    brsstrcat(ADR(StruktNovehoNazvuSuboru.CAS),ADR(Sekunda_STR));

    //Kód modelu//
    StruktNovehoNazvuSuboru.SERIAL:= FTP_CAM17.INPUTS.QRkodPowerCP;

    //Index fotky//
    StruktNovehoNazvuSuboru.INDEX:= FTP_CAM17.INPUTS.IndexFotky;

    //Result fotky//
    StruktNovehoNazvuSuboru.RESULT:= FTP_CAM17.INPUTS.Result;

	//Prípona súboru//
	IF TypFotky_BMP THEN
		StruktNovehoNazvuSuboru.Pripona:= '.bmp';
	ELSE
		StruktNovehoNazvuSuboru.Pripona:= '.jpg';
	END_IF

    //Mapovanie premenných//
    FTP_CAM17.STATUS.AdresarPrazdny:= AdresarPrazdny;

	CASE SC_Devlink.Step OF

		0:
			SC_Devlink.StepName:= '0 - Nulovanie';
			FTP_CAM17.STATUS.KomunikaciaError:= FALSE;
			FTP_CAM17.STATUS.KomunikaciaUkoncena:= FALSE;
			PocetHladaniFotky:= 0;
            AdresarPrazdny:= FALSE;
            PocetNajdenychSuborov:= 0;
            PocetNajdenychAdresarov:= 0;
            PocetPremenovanychSuborov:= 0;
            PocetSkopirovanychSuborov:= 0;
            PocetVymazanychSuborov:= 0;
            i:= 0;
            PocetPokusov_FTP_KOM:= 0;
			PoruchaKomunikacie:= FALSE;
			DirInfo_0.enable:= FALSE;
			DirRead_0.enable:= FALSE;
			FileRename_0.enable:= FALSE;
			DirCreate_0.enable:= FALSE;
			DirInfo_0.enable:= FALSE;
			DirRead_0.enable:= FALSE;
			FileCopy_0.enable:= FALSE;
			FileDelete_0.enable:= FALSE;
			SC_Devlink.Step:= 1;

        1:
            SC_Devlink.StepName:= '1 - Rozhodnutie o cinnosti';
            IF FTP_CAM17.CMD.OdosliFotku THEN
                FTP_CAM17.STATUS.PopisPoruchy:= '';
                SC_Devlink.Step:= 15;
            ELSIF FTP_CAM17.CMD.VymazFotku THEN
                FTP_CAM17.STATUS.PopisPoruchy:= '';
                SC_Devlink.Step:= 153;
            END_IF

		15:
			SC_Devlink.StepName:= '15 - Odoslanie fotky, kontrola pripojenia na FTP server Panasonic';
			SC_Devlink.IdleTime.PT:= T#3s;
			SC_Devlink.AlarmTime.PT:= T#3s;

			IF Stav_PripojenieFTP_OK THEN
				SC_Devlink.ResetStep:= TRUE;
				SC_Devlink.Step:= 20;
			END_IF

        20:
            SC_Devlink.StepName:= '20 - Odoslanie fotky na server, nacitanie adresara kamery pred premenovanim';
            SC_Devlink.IdleTime.PT:= T#3s;
            SC_Devlink.AlarmTime.PT:= T#3s;

            DirInfo_0.enable:= TRUE;
            DirInfo_0.pDevice:= ADR('CAM17');
            DirInfo_0.pPath:= ADR('/');   //ak je nula tak číta všetky súbory a adresáre v koreni ak je "/Temp" tak číta všetky súbory a adresáre v adresári Temp//
            DirInfo_0();

            IF DirInfo_0.status = 0 THEN
                PocetNajdenychAdresarov:= DirInfo_0.dirnum;
                PocetNajdenychSuborov:= DirInfo_0.filenum;
                brsmemset(ADR(FileList[0]),0, SIZEOF(FileList));  //Vynulovanie pola stringov pre záznam adresárov a súborov
                SC_Devlink.ResetStep:= TRUE;
                SC_Devlink.Step:= 23;
            ELSIF DirInfo_0.status = 65535 THEN
                //BUSY//
            ELSIF DirInfo_0.status = 20723 THEN
                FTP_CAM17.STATUS.PopisPoruchy:= 'Porucha nacitania adresara kamery';
                Buffer_17.Hodnota:= DirInfo_0.status;
                Buffer_17.ZapisHodnotu:= TRUE;
                PoruchaKomunikacie:= TRUE;
                SC_Devlink.ResetStep:= TRUE;
                SC_Devlink.Step:= 100;
            ELSE
                FTP_CAM17.STATUS.PopisPoruchy:= 'Porucha nacitania adresara kamery';
                IF DirInfo_0.status = 20799 THEN
                    Buffer_17.Hodnota:= FileIoGetSysError();
                ELSE
                    Buffer_17.Hodnota:= DirInfo_0.status;
                END_IF
                Buffer_17.ZapisHodnotu:= TRUE;
                PoruchaKomunikacie:= TRUE;
                SC_Devlink.ResetStep:= TRUE;
                SC_Devlink.Step:= 100;
            END_IF

        23:
            SC_Devlink.StepName:= '23 - Odoslanie fotky na server, kontrola poctu najdenych suborov v adresari kamery';
            SC_Devlink.IdleTime.PT:= T#3s;
            SC_Devlink.AlarmTime.PT:= T#3s;

            IF PocetNajdenychSuborov > 0 THEN
                PocetHladaniFotky:= 0;
                SC_Devlink.ResetStep:= TRUE;
                SC_Devlink.Step:= 25;
            ELSIF PocetHladaniFotky < 100 THEN
                PocetHladaniFotky:= PocetHladaniFotky + 1;
                SC_Devlink.ResetStep:= TRUE;
                SC_Devlink.Step:= 20;
            ELSIF PocetHladaniFotky >= 100 THEN
                AdresarPrazdny:= TRUE;
                FTP_CAM17.STATUS.KomunikaciaUkoncena:= TRUE;
                SC_Devlink.ResetStep:= TRUE;
                SC_Devlink.Step:= 100;
            END_IF

        25:
            SC_Devlink.StepName:= '25 - Odoslanie fotky na server, zapis nazvou najdenych suborov do pola stringov';
            SC_Devlink.IdleTime.PT:= T#3s;
            SC_Devlink.AlarmTime.PT:= T#3s;

            DirRead_0.enable:= TRUE;
            DirRead_0.pDevice:= ADR('CAM17');
            DirRead_0.pPath:= ADR('/');   //ak je nula tak číta všetky súbory a adresáre v koreni ak je "/Temp" tak číta všetky súbory a adresáre v adresári Temp//
            DirRead_0.option:= fiFILE; //Zapíše súbory aj adresáre, ak je fiDIRECTORY zapíše len adresáre, ak je fiFILE tak zapíše len súbory//
            DirRead_0.entry:= i; //index zapisovania do pola//
            DirRead_0.pData:= ADR(ReadData);
            DirRead_0.data_len:= SIZEOF(ReadData);
            DirRead_0();

            IF DirRead_0.status = 0 THEN
                brsstrcpy(ADR(FileList[i]), ADR(ReadData.Filename[0])); //Uloženie názvou adresárov a súborov do pola stringov
				IF i< 100 THEN
					i:= i + 1;
				END_IF
            ELSIF DirRead_0.status = 20702 THEN
                i:= 0;
                SC_Devlink.ResetStep:= TRUE;
                SC_Devlink.Step:= 28;
            ELSIF DirRead_0.status = 65535 THEN
                //BUSY//
            ELSE
                FTP_CAM17.STATUS.PopisPoruchy:= 'Porucha zapisu suborov do pola';
                PoruchaKomunikacie:= TRUE;
                SC_Devlink.ResetStep:= TRUE;
                SC_Devlink.Step:= 100;
            END_IF

        28:
            SC_Devlink.StepName:= '28 - Odoslanie fotky na server, premenovanie fotky';
            SC_Devlink.IdleTime.PT:= T#3s;
            SC_Devlink.AlarmTime.PT:= T#3s;

            StaryNazovSuboru:= '';
            brsstrcat(ADR(StaryNazovSuboru),ADR('/'));
            brsstrcat(ADR(StaryNazovSuboru),ADR(FileList[i]));

            NovyNazovSuboru:= '';
            brsstrcat(ADR(NovyNazovSuboru),ADR('/'));
            brsstrcat(ADR(NovyNazovSuboru),ADR(StruktNovehoNazvuSuboru.DATUM));
            brsstrcat(ADR(NovyNazovSuboru),ADR('_'));
            brsstrcat(ADR(NovyNazovSuboru),ADR(StruktNovehoNazvuSuboru.CAS));
            brsstrcat(ADR(NovyNazovSuboru),ADR('_'));
            brsstrcat(ADR(NovyNazovSuboru),ADR(StruktNovehoNazvuSuboru.SERIAL));
            brsstrcat(ADR(NovyNazovSuboru),ADR('_'));
            brsstrcat(ADR(NovyNazovSuboru),ADR(StruktNovehoNazvuSuboru.INDEX));
            brsstrcat(ADR(NovyNazovSuboru),ADR('_'));
            brsstrcat(ADR(NovyNazovSuboru),ADR(StruktNovehoNazvuSuboru.RESULT));
            brsstrcat(ADR(NovyNazovSuboru),ADR(StruktNovehoNazvuSuboru.Pripona));

            FileRename_0.enable:= TRUE;
            FileRename_0.pDevice:= ADR('CAM17');
            FileRename_0.pName:= ADR(StaryNazovSuboru);
            FileRename_0.pNewName:= ADR(NovyNazovSuboru);
            FileRename_0();

            IF FileRename_0.status = 0 THEN
                SC_Devlink.ResetStep:= TRUE;
                SC_Devlink.Step:= 30;
            ELSIF FileRename_0.status = 65535 THEN
                //BUSY//
            ELSIF FileRename_0.status = 20705 THEN
                SC_Devlink.ResetStep:= TRUE;
                SC_Devlink.Step:= 30;
            ELSIF FileRename_0.status = 20708 THEN
                AdresarPrazdny:= TRUE;
                FTP_CAM17.STATUS.KomunikaciaUkoncena:= TRUE;
                SC_Devlink.ResetStep:= TRUE;
                SC_Devlink.Step:= 100;
			ELSE
                FTP_CAM17.STATUS.PopisPoruchy:= 'Porucha premenovania fotky';
                PoruchaKomunikacie:= TRUE;
                SC_Devlink.ResetStep:= TRUE;
                SC_Devlink.Step:= 100;
            END_IF

        30:
            SC_Devlink.StepName:= '30 - Odoslanie fotky na server, kontrola poctu premenovanych suborov';
            SC_Devlink.IdleTime.PT:= T#3s;
            SC_Devlink.AlarmTime.PT:= T#3s;

            IF NOT SC_Devlink.Switch1 THEN
                PocetPremenovanychSuborov:= PocetPremenovanychSuborov + 1;
                SC_Devlink.Switch1:= TRUE;
            END_IF

            IF PocetPremenovanychSuborov < PocetNajdenychSuborov THEN
               	IF i< 100 THEN
					i:= i + 1;
				END_IF
                SC_Devlink.ResetStep:= TRUE;
                SC_Devlink.Step:= 28;
            ELSE
                i:= 0;
                PocetNajdenychSuborov:= 0;
                PocetNajdenychAdresarov:= 0;
                SC_Devlink.ResetStep:= TRUE;
                SC_Devlink.Step:= 33;//33
            END_IF

        33: SC_Devlink.StepName:= '33 - Odoslanie fotky na server, vytvorenie adresara LINKA';
            SC_Devlink.IdleTime.PT:= T#3s;
            SC_Devlink.AlarmTime.PT:= T#3s;

            NazovAdresara_LINKA:= '';
            brsstrcat(ADR(NazovAdresara_LINKA),ADR('DesignMP'));
            brsstrcat(ADR(NazovAdresara_LINKA),ADR('/'));
            brsstrcat(ADR(NazovAdresara_LINKA),ADR(StruktNovehoNazvuAdresara.LINKA));

            DirCreate_0.enable:= TRUE;
            DirCreate_0.pDevice:= ADR('Panasonic');
            DirCreate_0.pName:= ADR(NazovAdresara_LINKA);
            DirCreate_0();

            IF DirCreate_0.status = 0 THEN
                SC_Devlink.ResetStep:= TRUE;
                SC_Devlink.Step:= 35;
            ELSIF DirCreate_0.status = 65535 THEN
                //BUSY//
            ELSIF DirCreate_0.status = 20725 THEN
                SC_Devlink.ResetStep:= TRUE;
                SC_Devlink.Step:= 35;
            ELSIF DirCreate_0.status = 20709 THEN
                //BUSY//
            ELSE
                FTP_CAM17.STATUS.PopisPoruchy:= 'Porucha vytvorenia adresara na FTP Panasonic';
                PoruchaKomunikacie:= TRUE;
                SC_Devlink.ResetStep:= TRUE;
                SC_Devlink.Step:= 100;
            END_IF

        35: SC_Devlink.StepName:= '35 - Odoslanie fotky na server, vytvorenie podadresara PRACOVISKO';
            SC_Devlink.IdleTime.PT:= T#3s;
            SC_Devlink.AlarmTime.PT:= T#3s;

            NazovPodAdresara_PRACOVISKO:= '';
            brsstrcat(ADR(NazovPodAdresara_PRACOVISKO),ADR(NazovAdresara_LINKA));
            brsstrcat(ADR(NazovPodAdresara_PRACOVISKO),ADR('/'));
            brsstrcat(ADR(NazovPodAdresara_PRACOVISKO),ADR(StruktNovehoNazvuAdresara.PRACOVISKO));

            DirCreate_0.enable:= TRUE;
            DirCreate_0.pDevice:= ADR('Panasonic');
            DirCreate_0.pName:= ADR(NazovPodAdresara_PRACOVISKO);
            DirCreate_0();

            IF DirCreate_0.status = 0 THEN
                SC_Devlink.ResetStep:= TRUE;
                SC_Devlink.Step:= 38;
            ELSIF DirCreate_0.status = 65535 THEN
                //BUSY//
            ELSIF DirCreate_0.status = 20725 THEN
                SC_Devlink.ResetStep:= TRUE;
                SC_Devlink.Step:= 38;
            ELSIF DirCreate_0.status = 20709 THEN
                //BUSY//
            ELSE
                FTP_CAM17.STATUS.PopisPoruchy:= 'Porucha vytvorenia adresara na FTP Panasonic';
                PoruchaKomunikacie:= TRUE;
                SC_Devlink.ResetStep:= TRUE;
                SC_Devlink.Step:= 100;
            END_IF

        38: SC_Devlink.StepName:= '38 - Odoslanie fotky na server, vytvorenie podadresara ROK';
            SC_Devlink.IdleTime.PT:= T#3s;
            SC_Devlink.AlarmTime.PT:= T#3s;

            NazovPodAdresara_ROK:= '';
            brsstrcat(ADR(NazovPodAdresara_ROK),ADR(NazovPodAdresara_PRACOVISKO));
            brsstrcat(ADR(NazovPodAdresara_ROK),ADR('/'));
            brsstrcat(ADR(NazovPodAdresara_ROK),ADR(StruktNovehoNazvuAdresara.ROK));

            DirCreate_0.enable:= TRUE;
            DirCreate_0.pDevice:= ADR('Panasonic');
            DirCreate_0.pName:= ADR(NazovPodAdresara_ROK);
            DirCreate_0();

            IF DirCreate_0.status = 0 THEN
                SC_Devlink.ResetStep:= TRUE;
                SC_Devlink.Step:= 40;
            ELSIF DirCreate_0.status = 65535 THEN
                //BUSY//
            ELSIF DirCreate_0.status = 20725 THEN
                SC_Devlink.ResetStep:= TRUE;
                SC_Devlink.Step:= 40;
            ELSIF DirCreate_0.status = 20709 THEN
                //BUSY//
            ELSE
                FTP_CAM17.STATUS.PopisPoruchy:= 'Porucha vytvorenia adresara na FTP Panasonic';
                PoruchaKomunikacie:= TRUE;
                SC_Devlink.ResetStep:= TRUE;
                SC_Devlink.Step:= 100;
            END_IF

        40: SC_Devlink.StepName:= '40 - Odoslanie fotky na server, vytvorenie podadresara DATUM';
            SC_Devlink.IdleTime.PT:= T#3s;
            SC_Devlink.AlarmTime.PT:= T#3s;

            NazovPodAdresara_DATUM:= '';
            brsstrcat(ADR(NazovPodAdresara_DATUM),ADR(NazovPodAdresara_ROK));
            brsstrcat(ADR(NazovPodAdresara_DATUM),ADR('/'));
            brsstrcat(ADR(NazovPodAdresara_DATUM),ADR(StruktNovehoNazvuAdresara.DATUM));

            DirCreate_0.enable:= TRUE;
            DirCreate_0.pDevice:= ADR('Panasonic');
            DirCreate_0.pName:= ADR(NazovPodAdresara_DATUM);
            DirCreate_0();

            IF DirCreate_0.status = 0 THEN
                SC_Devlink.ResetStep:= TRUE;
                SC_Devlink.Step:= 43;
            ELSIF DirCreate_0.status = 65535 THEN
                //BUSY//
            ELSIF DirCreate_0.status = 20725 THEN
                SC_Devlink.ResetStep:= TRUE;
                SC_Devlink.Step:= 43;
            ELSIF DirCreate_0.status = 20709 THEN
                //BUSY//
            ELSE
                FTP_CAM17.STATUS.PopisPoruchy:= 'Porucha vytvorenia adresara na FTP Panasonic';
                PoruchaKomunikacie:= TRUE;
                SC_Devlink.ResetStep:= TRUE;
                SC_Devlink.Step:= 100;
            END_IF

        43:	SC_Devlink.StepName:= '43 - Odoslanie fotky na server, nacitanie adresara pred kopirovanim fotiek na server Panasonic';
            SC_Devlink.IdleTime.PT:= T#3s;
            SC_Devlink.AlarmTime.PT:= T#3s;

            DirInfo_0.enable:= TRUE;
            DirInfo_0.pDevice:= ADR('CAM17');
            DirInfo_0.pPath:= ADR('/');   //ak je nula tak číta všetky súbory a adresáre v koreni ak je "/Temp" tak číta všetky súbory a adresáre v adresári Temp//
            DirInfo_0();

            IF DirInfo_0.status = 0 THEN
                PocetNajdenychAdresarov:= DirInfo_0.dirnum;
                PocetNajdenychSuborov:= DirInfo_0.filenum;
                brsmemset(ADR(FileList[0]),0, SIZEOF(FileList));  //Vynulovanie pola stringov pre záznam adresárov a súborov
                SC_Devlink.ResetStep:= TRUE;
                SC_Devlink.Step:= 45;
            ELSIF DirInfo_0.status = 65535 THEN
                //BUSY//
            ELSIF DirInfo_0.status = 20723 THEN
                FTP_CAM17.STATUS.PopisPoruchy:= 'Porucha nacitania adresara kamery';
                Buffer_17.Hodnota:= DirInfo_0.status;
                Buffer_17.ZapisHodnotu:= TRUE;
                PoruchaKomunikacie:= TRUE;
                SC_Devlink.ResetStep:= TRUE;
                SC_Devlink.Step:= 100;
            ELSE
                FTP_CAM17.STATUS.PopisPoruchy:= 'Porucha nacitania adresara kamery';
                IF DirInfo_0.status = 20799 THEN
                    Buffer_17.Hodnota:= FileIoGetSysError();
                ELSE
                    Buffer_17.Hodnota:= DirInfo_0.status;
                END_IF
                Buffer_17.ZapisHodnotu:= TRUE;
                PoruchaKomunikacie:= TRUE;
                SC_Devlink.ResetStep:= TRUE;
                SC_Devlink.Step:= 100;
            END_IF

        45: SC_Devlink.StepName:= '45 - Odoslanie fotky na server, zapis nazvou najdenych suborov do pola stringov';
            SC_Devlink.IdleTime.PT:= T#3s;
            SC_Devlink.AlarmTime.PT:= T#3s;

            DirRead_0.enable:= TRUE;
            DirRead_0.pDevice:= ADR('CAM17');
            DirRead_0.pPath:= ADR('/');   //ak je nula tak číta všetky súbory a adresáre v koreni ak je "/Temp" tak číta všetky súbory a adresáre v adresári Temp//
            DirRead_0.option:= fiFILE; //Zapíše súbory aj adresáre, ak je fiDIRECTORY zapíše len adresáre, ak je fiFILE tak zapíše len súbory//
            DirRead_0.entry:= i; //index zapisovania do pola//
            DirRead_0.pData:= ADR(ReadData);
            DirRead_0.data_len:= SIZEOF(ReadData);
            DirRead_0();

            IF DirRead_0.status = 0 THEN
                brsstrcpy(ADR(FileList[i]), ADR(ReadData.Filename[0])); //Uloženie názvou adresárov a súborov do pola stringov
				IF i< 100 THEN
					i:= i + 1;
				END_IF
            ELSIF DirRead_0.status = 20702 THEN
                i:= 0;
                SC_Devlink.ResetStep:= TRUE;
                SC_Devlink.Step:= 47;
            ELSIF DirRead_0.status = 65535 THEN
                //BUSY//
            ELSE
                FTP_CAM17.STATUS.PopisPoruchy:= 'Porucha zapisu najdenych suborov do pola';
                PoruchaKomunikacie:= TRUE;
                SC_Devlink.ResetStep:= TRUE;
                SC_Devlink.Step:= 100;
            END_IF

		47:
			SC_Devlink.StepName:= '47 - Odoslanie fotky na server, vytvorenie cesty pre kopírovanie suboruk fotky na server Panasonic';
			SC_Devlink.IdleTime.PT:= T#3s;
			SC_Devlink.AlarmTime.PT:= T#3s;

			ZdrojKopirovaniaSuboru:= '';
			brsstrcat(ADR(ZdrojKopirovaniaSuboru),ADR('/'));
			brsstrcat(ADR(ZdrojKopirovaniaSuboru),ADR(ReadData.Filename));

			CielKopirovaniaSuboru:= '';
			brsstrcat(ADR(CielKopirovaniaSuboru),ADR(NazovPodAdresara_DATUM));
			brsstrcat(ADR(CielKopirovaniaSuboru),ADR('/'));
			brsstrcat(ADR(CielKopirovaniaSuboru),ADR(ReadData.Filename));

			SC_Devlink.ResetStep:= TRUE;
			SC_Devlink.Step:= 48;

        48: SC_Devlink.StepName:= '48 - Odoslanie fotky na server, kopirovanie fotky na server Panasonic';
            SC_Devlink.IdleTime.PT:= T#3s;
            SC_Devlink.AlarmTime.PT:= T#3s;

			FileCopy_0.enable:= TRUE;
			FileCopy_0.pSrcDev:= ADR('CAM17'); //Zdrojové zariadenie od kial sa kopíruje
			FileCopy_0.pSrc:= ADR(ZdrojKopirovaniaSuboru);
			FileCopy_0.pDestDev:= ADR('Panasonic'); //Cielové zariadenie kam sa má súbor skopírovať
			FileCopy_0.pDest:= ADR(CielKopirovaniaSuboru);
			FileCopy_0.option := fiOVERWRITE;
			FileCopy_0();

            IF FileCopy_0.status = 0 THEN
                SC_Devlink.ResetStep:= TRUE;
                SC_Devlink.Step:= 50;
            ELSIF FileCopy_0.status = 65535 THEN
                //BUSY//
            ELSIF FileCopy_0.status = 20705 THEN
                SC_Devlink.ResetStep:= TRUE;
				SC_Devlink.Step:= 50;
			ELSIF FileCopy_0.status = 20799 THEN
				SC_Devlink.ResetStep:= TRUE;
				SC_Devlink.Step:= 50;
            ELSIF FileCopy_0.status = 20708 THEN
                AdresarPrazdny:= TRUE;
                FTP_CAM17.STATUS.KomunikaciaUkoncena:= TRUE;
                SC_Devlink.ResetStep:= TRUE;
                SC_Devlink.Step:= 100;
            ELSE
                FTP_CAM17.STATUS.PopisPoruchy:= 'Porucha kopirovania fotky na FTP Panasonic';
                PoruchaKomunikacie:= TRUE;
                SC_Devlink.ResetStep:= TRUE;
                SC_Devlink.Step:= 100;
            END_IF

        50: SC_Devlink.StepName:= '50 - Odoslanie fotky na server, kontrola poctu skopirovanych suborov';
            SC_Devlink.IdleTime.PT:= T#3s;
            SC_Devlink.AlarmTime.PT:= T#3s;

            IF NOT SC_Devlink.Switch1 THEN
                PocetSkopirovanychSuborov:= PocetSkopirovanychSuborov + 1;
                SC_Devlink.Switch1:= TRUE;
            END_IF

            IF PocetSkopirovanychSuborov < PocetNajdenychSuborov THEN
                IF i< 100 THEN
					i:= i + 1;
				END_IF
                SC_Devlink.ResetStep:= TRUE;
                SC_Devlink.Step:= 48;
            ELSE
                i:= 0;
                PocetNajdenychSuborov:= 0;
                PocetNajdenychAdresarov:= 0;
                SC_Devlink.ResetStep:= TRUE;
                SC_Devlink.Step:= 60;
            END_IF

        60:
            SC_Devlink.StepName:= '60 - Odoslanie fotky na server, nacitanie adresara kamery pred vymazanim';
            SC_Devlink.IdleTime.PT:= T#3s;
            SC_Devlink.AlarmTime.PT:= T#3s;

            DirInfo_0.enable:= TRUE;
            DirInfo_0.pDevice:= ADR('CAM17');
            DirInfo_0.pPath:= ADR('/');   //ak je nula tak číta všetky súbory a adresáre v koreni ak je "/Temp" tak číta všetky súbory a adresáre v adresári Temp//
            DirInfo_0();

            IF DirInfo_0.status = 0 THEN
                PocetNajdenychAdresarov:= DirInfo_0.dirnum;
                PocetNajdenychSuborov:= DirInfo_0.filenum;
                brsmemset(ADR(FileList[0]),0, SIZEOF(FileList));  //Vynulovanie pola stringov pre záznam adresárov a súborov
                SC_Devlink.Step:= 63;
            ELSIF DirInfo_0.status = 65535 THEN
                //BUSY//
            ELSIF DirInfo_0.status = 20723 THEN
                FTP_CAM17.STATUS.PopisPoruchy:= 'Porucha nacitania adresara kamery';
                Buffer_17.Hodnota:= DirInfo_0.status;
                Buffer_17.ZapisHodnotu:= TRUE;
                PoruchaKomunikacie:= TRUE;
                SC_Devlink.ResetStep:= TRUE;
                SC_Devlink.Step:= 100;
            ELSE
                FTP_CAM17.STATUS.PopisPoruchy:= 'Porucha nacitania adresara kamery';
                IF DirInfo_0.status = 20799 THEN
                    Buffer_17.Hodnota:= FileIoGetSysError();
                ELSE
                    Buffer_17.Hodnota:= DirInfo_0.status;
                END_IF
                Buffer_17.ZapisHodnotu:= TRUE;
                PoruchaKomunikacie:= TRUE;
                SC_Devlink.ResetStep:= TRUE;
                SC_Devlink.Step:= 100;
            END_IF

        63: SC_Devlink.StepName:= '63 - Odoslanie fotky na server, zapis nazvou najdenych suborov do pola stringov';
            SC_Devlink.IdleTime.PT:= T#3s;
            SC_Devlink.AlarmTime.PT:= T#3s;

            DirRead_0.enable:= TRUE;
            DirRead_0.pDevice:= ADR('CAM17');
            DirRead_0.pPath:= ADR('/');   //ak je nula tak číta všetky súbory a adresáre v koreni ak je "/Temp" tak číta všetky súbory a adresáre v adresári Temp//
            DirRead_0.option:= fiFILE; //Zapíše súbory aj adresáre, ak je fiDIRECTORY zapíše len adresáre, ak je fiFILE tak zapíše len súbory//
            DirRead_0.entry:= i; //index zapisovania do pola//
            DirRead_0.pData:= ADR(ReadData);
            DirRead_0.data_len:= SIZEOF(ReadData);
            DirRead_0();

            IF DirRead_0.status = 0 THEN
                brsstrcpy(ADR(FileList[i]), ADR(ReadData.Filename[0])); //Uloženie názvou adresárov a súborov do pola stringov
				IF i< 100 THEN
					i:= i + 1;
				END_IF
            ELSIF DirRead_0.status = 20702 THEN
                i:= 0;
                SC_Devlink.ResetStep:= TRUE;
                SC_Devlink.Step:= 65;
            ELSIF DirRead_0.status = 65535 THEN
                //BUSY//
            ELSE
                FTP_CAM17.STATUS.PopisPoruchy:= 'Porucha zapisu najdenych suborov do pola';
                PoruchaKomunikacie:= TRUE;
                SC_Devlink.ResetStep:= TRUE;
                SC_Devlink.Step:= 100;
            END_IF

        65: SC_Devlink.StepName:= '65 - Odoslanie fotky na server, vymazanie suboru';
            SC_Devlink.IdleTime.PT:= T#3s;
            SC_Devlink.AlarmTime.PT:= T#3s;

            ZdrojKopirovaniaSuboru:= '';
            brsstrcat(ADR(ZdrojKopirovaniaSuboru),ADR('/'));
            brsstrcat(ADR(ZdrojKopirovaniaSuboru),ADR(FileList[i]));

            FileDelete_0.enable:= TRUE;
            FileDelete_0.pDevice:= ADR('CAM17');
            FileDelete_0.pName:= ADR(ZdrojKopirovaniaSuboru);
            FileDelete_0();

            IF FileDelete_0.status = 0 THEN
                SC_Devlink.ResetStep:= TRUE;
                SC_Devlink.Step:= 68;
            ELSIF FileDelete_0.status = 65535 THEN
                //BUSY//
            ELSIF FileDelete_0.status = 20708 THEN
                SC_Devlink.ResetStep:= TRUE;
                SC_Devlink.Step:= 68;
            ELSE
                FTP_CAM17.STATUS.PopisPoruchy:= 'Porucha vymazania fotky v adresari kamery';
                PoruchaKomunikacie:= TRUE;
                SC_Devlink.ResetStep:= TRUE;
                SC_Devlink.Step:= 100;
            END_IF

        68:	SC_Devlink.StepName:= '68 - Odoslanie fotky na server, kontrola poctu vymazanych suborov';
            SC_Devlink.IdleTime.PT:= T#3s;
            SC_Devlink.AlarmTime.PT:= T#3s;

            IF NOT SC_Devlink.Switch1 THEN
                PocetVymazanychSuborov:= PocetVymazanychSuborov + 1;
                SC_Devlink.Switch1:= TRUE;
            END_IF

            IF PocetVymazanychSuborov < PocetNajdenychSuborov THEN
                IF i< 100 THEN
					i:= i + 1;
				END_IF
                SC_Devlink.ResetStep:= TRUE;
                SC_Devlink.Step:= 65;
            ELSE
                i:= 0;
                PocetNajdenychSuborov:= 0;
                PocetNajdenychAdresarov:= 0;
                CAM17_PocetFotiek:= 0;
				FTP_CAM17.STATUS.KomunikaciaUkoncena:= TRUE;
                SC_Devlink.ResetStep:= TRUE;
                SC_Devlink.Step:= 100;
            END_IF

        100:
            SC_Devlink.StepName:= '100 - Odoslanie fotky, cakam na zrusenie prikazu odosli fotku';
            SC_Devlink.IdleTime.PT:= T#1s;
            SC_Devlink.AlarmTime.PT:= T#3s;

            SC_Devlink.IdleTime.IN:= TRUE;

            IF PoruchaKomunikacie AND SC_Devlink.IdleTime.Q AND PocetPokusov_FTP_KOM < 3 THEN
                PocetPokusov_FTP_KOM:= PocetPokusov_FTP_KOM + 1;
                PoruchaKomunikacie:= FALSE;
                i:= 0;
                PocetNajdenychSuborov:= 0;
                PocetNajdenychAdresarov:= 0;
                SC_Devlink.ResetStep:= TRUE;
                SC_Devlink.Step:= 1;
            ELSIF PoruchaKomunikacie AND PocetPokusov_FTP_KOM >= 3 THEN
                FTP_CAM17.STATUS.KomunikaciaError:= TRUE;
            END_IF

            IF NOT FTP_CAM17.CMD.OdosliFotku THEN
                SC_Devlink.ResetStep:= TRUE;
                SC_Devlink.Step:= 0;
            END_IF

            //**************************************Vymazanie fotky*************************************************//

		153:
			SC_Devlink.StepName:= '153 - Vymazanie fotky, nacitanie adresara kamery pred vymazanim';
			SC_Devlink.IdleTime.PT:= T#3s;
			SC_Devlink.AlarmTime.PT:= T#3s;

			DirInfo_0.enable:= TRUE;
			DirInfo_0.pDevice:= ADR('CAM17');
			DirInfo_0.pPath:= ADR('/');   //ak je nula tak číta všetky súbory a adresáre v koreni ak je "/Temp" tak číta všetky súbory a adresáre v adresári Temp//
			DirInfo_0();

			IF DirInfo_0.status = 0 THEN
				PocetNajdenychAdresarov:= DirInfo_0.dirnum;
				PocetNajdenychSuborov:= DirInfo_0.filenum;
				brsmemset(ADR(FileList[0]),0, SIZEOF(FileList));  //Vynulovanie pola stringov pre záznam adresárov a súborov
				SC_Devlink.Step:= 155;
			ELSIF DirInfo_0.status = 65535 THEN
				//BUSY//
			ELSIF DirInfo_0.status = 20723 THEN
				FTP_CAM17.STATUS.PopisPoruchy:= 'Porucha nacitania adresara kamery';
				Buffer_17.Hodnota:= DirInfo_0.status;
				Buffer_17.ZapisHodnotu:= TRUE;
				PoruchaKomunikacie:= TRUE;
				SC_Devlink.ResetStep:= TRUE;
				SC_Devlink.Step:= 200;
			ELSE
				FTP_CAM17.STATUS.PopisPoruchy:= 'Porucha nacitania adresara kamery';
				IF DirInfo_0.status = 20799 THEN
					Buffer_17.Hodnota:= FileIoGetSysError();
				ELSE
					Buffer_17.Hodnota:= DirInfo_0.status;
				END_IF
				Buffer_17.ZapisHodnotu:= TRUE;
				PoruchaKomunikacie:= TRUE;
				SC_Devlink.ResetStep:= TRUE;
				SC_Devlink.Step:= 200;
			END_IF

		155: SC_Devlink.StepName:= '155 - Vymazanie fotky, zapis nazvou najdenych suborov do pola stringov';
			SC_Devlink.IdleTime.PT:= T#3s;
			SC_Devlink.AlarmTime.PT:= T#3s;

			DirRead_0.enable:= TRUE;
			DirRead_0.pDevice:= ADR('CAM17');
			DirRead_0.pPath:= ADR('/');   //ak je nula tak číta všetky súbory a adresáre v koreni ak je "/Temp" tak číta všetky súbory a adresáre v adresári Temp//
			DirRead_0.option:= fiFILE; //Zapíše súbory aj adresáre, ak je fiDIRECTORY zapíše len adresáre, ak je fiFILE tak zapíše len súbory//
			DirRead_0.entry:= i; //index zapisovania do pola//
			DirRead_0.pData:= ADR(ReadData);
			DirRead_0.data_len:= SIZEOF(ReadData);
			DirRead_0();

			IF DirRead_0.status = 0 THEN
				brsstrcpy(ADR(FileList[i]), ADR(ReadData.Filename[0])); //Uloženie názvou adresárov a súborov do pola stringov
				IF i< 100 THEN
					i:= i + 1;
				END_IF
			ELSIF DirRead_0.status = 20702 THEN
				i:= 0;
				SC_Devlink.ResetStep:= TRUE;
				SC_Devlink.Step:= 158;
			ELSIF DirRead_0.status = 65535 THEN
				//BUSY//
			ELSE
				FTP_CAM17.STATUS.PopisPoruchy:= 'Porucha zapisu najdenych suborov do pola';
				PoruchaKomunikacie:= TRUE;
				SC_Devlink.ResetStep:= TRUE;
				SC_Devlink.Step:= 200;
			END_IF

		158: SC_Devlink.StepName:= '158 - Vymazanie fotky, vymazanie suboru';
			SC_Devlink.IdleTime.PT:= T#3s;
			SC_Devlink.AlarmTime.PT:= T#3s;

			ZdrojKopirovaniaSuboru:= '';
			brsstrcat(ADR(ZdrojKopirovaniaSuboru),ADR('/'));
			brsstrcat(ADR(ZdrojKopirovaniaSuboru),ADR(FileList[i]));

			FileDelete_0.enable:= TRUE;
			FileDelete_0.pDevice:= ADR('CAM17');
			FileDelete_0.pName:= ADR(ZdrojKopirovaniaSuboru);
			FileDelete_0();

			IF FileDelete_0.status = 0 THEN
				SC_Devlink.ResetStep:= TRUE;
				SC_Devlink.Step:= 160;
			ELSIF FileDelete_0.status = 65535 THEN
				//BUSY//
            ELSIF FileDelete_0.status = 20708 THEN
                SC_Devlink.ResetStep:= TRUE;
                SC_Devlink.Step:= 160;
            ELSE
                FTP_CAM17.STATUS.PopisPoruchy:= 'Porucha vymazania fotky v adresari kamery';
                PoruchaKomunikacie:= TRUE;
                SC_Devlink.ResetStep:= TRUE;
                SC_Devlink.Step:= 200;
            END_IF

        160:	SC_Devlink.StepName:= '160 - Vymazanie fotky, kontrola poctu vymazanych suborov';
            SC_Devlink.IdleTime.PT:= T#3s;
            SC_Devlink.AlarmTime.PT:= T#3s;

            IF NOT SC_Devlink.Switch1 THEN
                PocetVymazanychSuborov:= PocetVymazanychSuborov + 1;
                SC_Devlink.Switch1:= TRUE;
            END_IF

            IF PocetVymazanychSuborov < PocetNajdenychSuborov THEN
                IF i< 100 THEN
					i:= i + 1;
				END_IF
                SC_Devlink.ResetStep:= TRUE;
                SC_Devlink.Step:= 158;
            ELSE
                i:= 0;
                PocetNajdenychSuborov:= 0;
                PocetNajdenychAdresarov:= 0;
                CAM17_PocetFotiek:= 0;
				FTP_CAM17.STATUS.KomunikaciaUkoncena:= TRUE;
                SC_Devlink.ResetStep:= TRUE;
                SC_Devlink.Step:= 200;
            END_IF

        200:
            SC_Devlink.StepName:= '200 - Vymazanie fotky, cakam na zrusenie prikazu odosli fotku';
            SC_Devlink.IdleTime.PT:= T#1s;
            SC_Devlink.AlarmTime.PT:= T#3s;

            SC_Devlink.IdleTime.IN:= TRUE;

            IF PoruchaKomunikacie AND SC_Devlink.IdleTime.Q AND PocetPokusov_FTP_KOM < 3 THEN
                PocetPokusov_FTP_KOM:= PocetPokusov_FTP_KOM + 1;
                PoruchaKomunikacie:= FALSE;
                i:= 0;
                PocetNajdenychSuborov:= 0;
                PocetNajdenychAdresarov:= 0;
                SC_Devlink.ResetStep:= TRUE;
                SC_Devlink.Step:= 1;
            ELSIF PoruchaKomunikacie AND PocetPokusov_FTP_KOM >= 3 THEN
                FTP_CAM17.STATUS.KomunikaciaError:= TRUE;
            END_IF

            IF NOT FTP_CAM17.CMD.VymazFotku THEN
                SC_Devlink.ResetStep:= TRUE;
                SC_Devlink.Step:= 0;
            END_IF

    END_CASE

END_PROGRAM

PROGRAM _EXIT
	(* Insert code here *)

END_PROGRAM
```

#### Variables.var - Local variables
```iecst
VAR
	SC_Devlink : SequenceControlTyp;
	DirInfo_0 : DirInfo;
	DirRead_0 : DirRead;
	FileRename_0 : FileRename;
	FileDelete_0 : FileDelete;
	FileCopy_0 : FileCopy;
	DirCreate_0 : DirCreate;
	i : UDINT;
	FileList : ARRAY[0..100] OF STRING[100];
	ReadData : fiDIR_READ_DATA; (*data-structure for command bDirRead*)
	PocetNajdenychAdresarov : UDINT;
	PocetNajdenychSuborov : UDINT;
	PocetPremenovanychSuborov : UDINT;
	PocetSkopirovanychSuborov : UDINT;
	PocetVymazanychSuborov : UDINT;
	StaryNazovSuboru : STRING[200];
	NovyNazovSuboru : STRING[200];
	ZdrojKopirovaniaSuboru : STRING[200];
	CielKopirovaniaSuboru : STRING[200];
	AdresarPrazdny : BOOL;
	StruktNovehoNazvuSuboru : StrukturaNovehoNazvuSuboru_typ;
	StruktNovehoNazvuAdresara : StrukturaNovehoNazvuAdresara_typ;
	NazovAdresara_LINKA : STRING[50];
	NazovPodAdresara_PRACOVISKO : STRING[50];
	NazovPodAdresara_ROK : STRING[50];
	NazovPodAdresara_DATUM : STRING[50];
	PocetHladaniFotky : UDINT;
	PocetPokusov_FTP_KOM : USINT;
	PoruchaKomunikacie : BOOL;
END_VAR
```

### Program Logical/OdosielanieFotiek/DevlinkFTP (IEC)

#### Main.st - Init, cyclic, exit code
```iecst
PROGRAM _INIT
	(* Insert code here *)

END_PROGRAM

PROGRAM _CYCLIC

	//Volanie funkcie SequenceControl//
	SequenceControl(SC:= SC_DevlinkFTP);

	CASE SC_DevlinkFTP.Step OF

		0:
			SC_DevlinkFTP.StepName:= '0 - Nulovanie';
			SC_DevlinkFTP.IdleTime.PT:= T#3s;
			SC_DevlinkFTP.AlarmTime.PT:= T#3s;

			DevLink_0.enable:= FALSE;
			DevUnlink_0.enable:= FALSE;
			Stav_PripojenieFTP_OK:= FALSE;
			OdpojServerFTP:= FALSE;

			SC_DevlinkFTP.ResetStep:= TRUE;
			SC_DevlinkFTP.Step:= 1;

		1:
			SC_DevlinkFTP.StepName:= '1 - Pripojenie na FTP server Panasonic';
			SC_DevlinkFTP.IdleTime.PT:= T#3s;
			SC_DevlinkFTP.AlarmTime.PT:= T#3s;

			DevLink_0.enable:= TRUE;
			DevLink_0.pDevice:= ADR('Panasonic');
			DevLink_0.pParam:= ADR('/SIP=192.168.100.164 /PROTOCOL=ftp /USER=designMP /PASSWORD=Ftp4PAN2020');
			(*DevLink_0.pParam:= ADR('/SIP=10.128.149.2 /PROTOCOL=ftp /USER=designMP /PASSWORD=Ftp4PAN2020');*)
			DevLink_0();

			IF DevLink_0.status = 0 THEN
				ID_Adresara:= DevLink_0.handle;
				Stav_PripojenieFTP_OK:= TRUE;
				SC_DevlinkFTP.ResetStep:= TRUE;
				SC_DevlinkFTP.Step:= 10;
			ELSIF DevLink_0.status = 20730 THEN
				ID_Adresara:= DevLink_0.handle;
				Stav_PripojenieFTP_OK:= TRUE;
				SC_DevlinkFTP.ResetStep:= TRUE;
				SC_DevlinkFTP.Step:= 10;
			ELSIF DevLink_0.status = 65535 THEN
				//BUSY//
			END_IF

		10:
			SC_DevlinkFTP.StepName:= '10 - Cakam na odpojenie od FTP servera Panasonic';
			SC_DevlinkFTP.IdleTime.PT:= T#3s;
			SC_DevlinkFTP.AlarmTime.PT:= T#3s;

			IF OdpojServerFTP THEN
				SC_DevlinkFTP.ResetStep:= TRUE;
				SC_DevlinkFTP.Step:= 15;
			END_IF

		15: SC_DevlinkFTP.StepName:= '15 - Odpojenie od FTP servera Panasonic';
			SC_DevlinkFTP.IdleTime.PT:= T#3s;
			SC_DevlinkFTP.AlarmTime.PT:= T#3s;

			DevUnlink_0.enable:= TRUE;
			DevUnlink_0.handle:= ID_Adresara;
			DevUnlink_0();

			IF DevUnlink_0.status = 0 THEN
				SC_DevlinkFTP.ResetStep:= TRUE;
				SC_DevlinkFTP.Step:= 0;
			ELSIF DevUnlink_0.status = 20798 THEN
				SC_DevlinkFTP.ResetStep:= TRUE;
				SC_DevlinkFTP.Step:= 0;
			ELSIF DevUnlink_0.status = 20731 THEN
				SC_DevlinkFTP.ResetStep:= TRUE;
				SC_DevlinkFTP.Step:= 0;
			ELSIF DevUnlink_0.status = 65535 THEN
				//BUSY//
			END_IF

	END_CASE

END_PROGRAM

PROGRAM _EXIT
	(* Insert code here *)

END_PROGRAM
```

#### Variables.var - Local variables
```iecst
VAR
	SC_DevlinkFTP : SequenceControlTyp := (0);
	ID_Adresara : UDINT;
	DevLink_0 : DevLink;
	DevUnlink_0 : DevUnlink;
END_VAR
```

### UkladacieBufferyGlobal.typ - Global data types
```iecst
TYPE
	UkladaciBuffer_typ : 	STRUCT
		Pole : ARRAY[0..100]OF REAL;
		Index : UINT;
		ZapisHodnotu : BOOL;
		ResetBufferu : BOOL;
		Hodnota : REAL;
	END_STRUCT;
END_TYPE
```

### UkladacieBufferyGlobal.var - Global variables
```iecst
VAR RETAIN
	Buffer_1 : UkladaciBuffer_typ;
	Buffer_2 : UkladaciBuffer_typ;
	Buffer_3 : UkladaciBuffer_typ;
	Buffer_4 : UkladaciBuffer_typ;
	Buffer_5 : UkladaciBuffer_typ;
	Buffer_6 : UkladaciBuffer_typ;
	Buffer_7 : UkladaciBuffer_typ;
	Buffer_8 : UkladaciBuffer_typ;
	Buffer_9 : UkladaciBuffer_typ;
	Buffer_10 : UkladaciBuffer_typ;
	Buffer_11 : UkladaciBuffer_typ;
	Buffer_12 : UkladaciBuffer_typ;
	Buffer_13 : UkladaciBuffer_typ;
	Buffer_14 : UkladaciBuffer_typ;
	Buffer_15 : UkladaciBuffer_typ;
	Buffer_16 : UkladaciBuffer_typ;
	Buffer_17 : UkladaciBuffer_typ;
	Buffer_18 : UkladaciBuffer_typ;
	Buffer_19 : UkladaciBuffer_typ;
	Buffer_20 : UkladaciBuffer_typ;
END_VAR
```

### Program Logical/UkladacieBuffery/UkladacieBuffery (IEC)

#### Main.st - Init, cyclic, exit code
```iecst
PROGRAM _INIT
	(* Insert code here *)

END_PROGRAM

PROGRAM _CYCLIC

    //*********************************************Buffer 1****************************************************//
    //Resetovanie//
    IF Buffer_1.ResetBufferu THEN
        brsmemset(ADR(Buffer_1.Pole),0,SIZEOF(Buffer_1.Pole));
        Buffer_1.Index:= 0;
        Buffer_1.ResetBufferu:= FALSE;
    END_IF

    //Zápis do buffera//
    IF Buffer_1.ZapisHodnotu THEN
        Buffer_1.Pole[Buffer_1.Index]:= Buffer_1.Hodnota;
        IF Buffer_1.Index < 100 THEN
            Buffer_1.Index:= Buffer_1.Index + 1;
        ELSE
            Buffer_1.Index:= 0;
        END_IF
        Buffer_1.ZapisHodnotu:= FALSE;
    END_IF

    //*********************************************Buffer 2****************************************************//
    //Resetovanie//
    IF Buffer_2.ResetBufferu THEN
        brsmemset(ADR(Buffer_2.Pole),0,SIZEOF(Buffer_2.Pole));
        Buffer_2.Index:= 0;
        Buffer_2.ResetBufferu:= FALSE;
    END_IF

    //Zápis do buffera//
    IF Buffer_2.ZapisHodnotu THEN
        Buffer_2.Pole[Buffer_2.Index]:= Buffer_2.Hodnota;
        IF Buffer_2.Index < 100 THEN
            Buffer_2.Index:= Buffer_2.Index + 1;
        ELSE
            Buffer_2.Index:= 0;
        END_IF
        Buffer_2.ZapisHodnotu:= FALSE;
    END_IF

    //*********************************************Buffer 3****************************************************//
    //Resetovanie//
    IF Buffer_3.ResetBufferu THEN
        brsmemset(ADR(Buffer_3.Pole),0,SIZEOF(Buffer_3.Pole));
        Buffer_3.Index:= 0;
        Buffer_3.ResetBufferu:= FALSE;
    END_IF

    //Zápis do buffera//
    IF Buffer_3.ZapisHodnotu THEN
        Buffer_3.Pole[Buffer_3.Index]:= Buffer_3.Hodnota;
        IF Buffer_3.Index < 100 THEN
            Buffer_3.Index:= Buffer_3.Index + 1;
        ELSE
            Buffer_3.Index:= 0;
        END_IF
        Buffer_3.ZapisHodnotu:= FALSE;
    END_IF

    //*********************************************Buffer 4****************************************************//
    //Resetovanie//
    IF Buffer_4.ResetBufferu THEN
        brsmemset(ADR(Buffer_4.Pole),0,SIZEOF(Buffer_4.Pole));
        Buffer_4.Index:= 0;
        Buffer_4.ResetBufferu:= FALSE;
    END_IF

    //Zápis do buffera//
    IF Buffer_4.ZapisHodnotu THEN
        Buffer_4.Pole[Buffer_4.Index]:= Buffer_4.Hodnota;
        IF Buffer_4.Index < 100 THEN
            Buffer_4.Index:= Buffer_4.Index + 1;
        ELSE
            Buffer_4.Index:= 0;
        END_IF
        Buffer_4.ZapisHodnotu:= FALSE;
    END_IF

    //*********************************************Buffer 5****************************************************//
    //Resetovanie//
    IF Buffer_5.ResetBufferu THEN
        brsmemset(ADR(Buffer_5.Pole),0,SIZEOF(Buffer_5.Pole));
        Buffer_5.Index:= 0;
        Buffer_5.ResetBufferu:= FALSE;
    END_IF

    //Zápis do buffera//
    IF Buffer_5.ZapisHodnotu THEN
        Buffer_5.Pole[Buffer_5.Index]:= Buffer_5.Hodnota;
        IF Buffer_5.Index < 100 THEN
            Buffer_5.Index:= Buffer_5.Index + 1;
        ELSE
            Buffer_5.Index:= 0;
        END_IF
        Buffer_5.ZapisHodnotu:= FALSE;
    END_IF

    //*********************************************Buffer 6****************************************************//
    //Resetovanie//
    IF Buffer_6.ResetBufferu THEN
        brsmemset(ADR(Buffer_6.Pole),0,SIZEOF(Buffer_6.Pole));
        Buffer_6.Index:= 0;
        Buffer_6.ResetBufferu:= FALSE;
    END_IF

    //Zápis do buffera//
    IF Buffer_6.ZapisHodnotu THEN
        Buffer_6.Pole[Buffer_6.Index]:= Buffer_6.Hodnota;
        IF Buffer_6.Index < 100 THEN
            Buffer_6.Index:= Buffer_6.Index + 1;
        ELSE
            Buffer_6.Index:= 0;
        END_IF
        Buffer_6.ZapisHodnotu:= FALSE;
    END_IF

    //*********************************************Buffer 7****************************************************//
    //Resetovanie//
    IF Buffer_7.ResetBufferu THEN
        brsmemset(ADR(Buffer_7.Pole),0,SIZEOF(Buffer_7.Pole));
        Buffer_7.Index:= 0;
        Buffer_7.ResetBufferu:= FALSE;
    END_IF

    //Zápis do buffera//
    IF Buffer_7.ZapisHodnotu THEN
        Buffer_7.Pole[Buffer_7.Index]:= Buffer_7.Hodnota;
        IF Buffer_7.Index < 100 THEN
            Buffer_7.Index:= Buffer_7.Index + 1;
        ELSE
            Buffer_7.Index:= 0;
        END_IF
        Buffer_7.ZapisHodnotu:= FALSE;
    END_IF

    //*********************************************Buffer 8****************************************************//
    //Resetovanie//
    IF Buffer_8.ResetBufferu THEN
        brsmemset(ADR(Buffer_8.Pole),0,SIZEOF(Buffer_8.Pole));
        Buffer_8.Index:= 0;
        Buffer_8.ResetBufferu:= FALSE;
    END_IF

    //Zápis do buffera//
    IF Buffer_8.ZapisHodnotu THEN
        Buffer_8.Pole[Buffer_8.Index]:= Buffer_8.Hodnota;
        IF Buffer_8.Index < 100 THEN
            Buffer_8.Index:= Buffer_8.Index + 1;
        ELSE
            Buffer_8.Index:= 0;
        END_IF
        Buffer_8.ZapisHodnotu:= FALSE;
    END_IF

    //*********************************************Buffer 9****************************************************//
    //Resetovanie//
    IF Buffer_9.ResetBufferu THEN
        brsmemset(ADR(Buffer_9.Pole),0,SIZEOF(Buffer_9.Pole));
        Buffer_9.Index:= 0;
        Buffer_9.ResetBufferu:= FALSE;
    END_IF

    //Zápis do buffera//
    IF Buffer_9.ZapisHodnotu THEN
        Buffer_9.Pole[Buffer_9.Index]:= Buffer_9.Hodnota;
        IF Buffer_9.Index < 100 THEN
            Buffer_9.Index:= Buffer_9.Index + 1;
        ELSE
            Buffer_9.Index:= 0;
        END_IF
        Buffer_9.ZapisHodnotu:= FALSE;
    END_IF

    //*********************************************Buffer 10****************************************************//
    //Resetovanie//
    IF Buffer_10.ResetBufferu THEN
        brsmemset(ADR(Buffer_10.Pole),0,SIZEOF(Buffer_10.Pole));
        Buffer_10.Index:= 0;
        Buffer_10.ResetBufferu:= FALSE;
    END_IF

    //Zápis do buffera//
    IF Buffer_10.ZapisHodnotu THEN
        Buffer_10.Pole[Buffer_10.Index]:= Buffer_10.Hodnota;
        IF Buffer_10.Index < 100 THEN
            Buffer_10.Index:= Buffer_10.Index + 1;
        ELSE
            Buffer_10.Index:= 0;
        END_IF
        Buffer_10.ZapisHodnotu:= FALSE;
    END_IF

    //*********************************************Buffer 11****************************************************//
    //Resetovanie//
    IF Buffer_11.ResetBufferu THEN
        brsmemset(ADR(Buffer_11.Pole),0,SIZEOF(Buffer_11.Pole));
        Buffer_11.Index:= 0;
        Buffer_11.ResetBufferu:= FALSE;
    END_IF

    //Zápis do buffera//
    IF Buffer_11.ZapisHodnotu THEN
        Buffer_11.Pole[Buffer_11.Index]:= Buffer_11.Hodnota;
        IF Buffer_11.Index < 100 THEN
            Buffer_11.Index:= Buffer_11.Index + 1;
        ELSE
            Buffer_11.Index:= 0;
        END_IF
        Buffer_11.ZapisHodnotu:= FALSE;
    END_IF

    //*********************************************Buffer 12****************************************************//
    //Resetovanie//
    IF Buffer_12.ResetBufferu THEN
        brsmemset(ADR(Buffer_12.Pole),0,SIZEOF(Buffer_12.Pole));
        Buffer_12.Index:= 0;
        Buffer_12.ResetBufferu:= FALSE;
    END_IF

    //Zápis do buffera//
    IF Buffer_12.ZapisHodnotu THEN
        Buffer_12.Pole[Buffer_12.Index]:= Buffer_12.Hodnota;
        IF Buffer_12.Index < 100 THEN
            Buffer_12.Index:= Buffer_12.Index + 1;
        ELSE
            Buffer_12.Index:= 0;
        END_IF
        Buffer_12.ZapisHodnotu:= FALSE;
    END_IF

    //*********************************************Buffer 13****************************************************//
    //Resetovanie//
    IF Buffer_13.ResetBufferu THEN
        brsmemset(ADR(Buffer_13.Pole),0,SIZEOF(Buffer_13.Pole));
        Buffer_13.Index:= 0;
        Buffer_13.ResetBufferu:= FALSE;
    END_IF

    //Zápis do buffera//
    IF Buffer_13.ZapisHodnotu THEN
        Buffer_13.Pole[Buffer_13.Index]:= Buffer_13.Hodnota;
        IF Buffer_13.Index < 100 THEN
            Buffer_13.Index:= Buffer_13.Index + 1;
        ELSE
            Buffer_13.Index:= 0;
        END_IF
        Buffer_13.ZapisHodnotu:= FALSE;
    END_IF

    //*********************************************Buffer 14****************************************************//
    //Resetovanie//
    IF Buffer_14.ResetBufferu THEN
        brsmemset(ADR(Buffer_14.Pole),0,SIZEOF(Buffer_14.Pole));
        Buffer_14.Index:= 0;
        Buffer_14.ResetBufferu:= FALSE;
    END_IF

    //Zápis do buffera//
    IF Buffer_14.ZapisHodnotu THEN
        Buffer_14.Pole[Buffer_14.Index]:= Buffer_14.Hodnota;
        IF Buffer_14.Index < 100 THEN
            Buffer_14.Index:= Buffer_14.Index + 1;
        ELSE
            Buffer_14.Index:= 0;
        END_IF
        Buffer_14.ZapisHodnotu:= FALSE;
    END_IF

    //*********************************************Buffer 15****************************************************//
    //Resetovanie//
    IF Buffer_15.ResetBufferu THEN
        brsmemset(ADR(Buffer_15.Pole),0,SIZEOF(Buffer_15.Pole));
        Buffer_15.Index:= 0;
        Buffer_15.ResetBufferu:= FALSE;
    END_IF

    //Zápis do buffera//
    IF Buffer_15.ZapisHodnotu THEN
        Buffer_15.Pole[Buffer_15.Index]:= Buffer_15.Hodnota;
        IF Buffer_15.Index < 100 THEN
            Buffer_15.Index:= Buffer_15.Index + 1;
        ELSE
            Buffer_15.Index:= 0;
        END_IF
        Buffer_15.ZapisHodnotu:= FALSE;
    END_IF

    //*********************************************Buffer 16****************************************************//
    //Resetovanie//
    IF Buffer_16.ResetBufferu THEN
        brsmemset(ADR(Buffer_16.Pole),0,SIZEOF(Buffer_16.Pole));
        Buffer_16.Index:= 0;
        Buffer_16.ResetBufferu:= FALSE;
    END_IF

    //Zápis do buffera//
    IF Buffer_16.ZapisHodnotu THEN
        Buffer_16.Pole[Buffer_16.Index]:= Buffer_16.Hodnota;
        IF Buffer_16.Index < 100 THEN
            Buffer_16.Index:= Buffer_16.Index + 1;
        ELSE
            Buffer_16.Index:= 0;
        END_IF
        Buffer_16.ZapisHodnotu:= FALSE;
    END_IF

    //*********************************************Buffer 17****************************************************//
    //Resetovanie//
    IF Buffer_17.ResetBufferu THEN
        brsmemset(ADR(Buffer_17.Pole),0,SIZEOF(Buffer_17.Pole));
        Buffer_17.Index:= 0;
        Buffer_17.ResetBufferu:= FALSE;
    END_IF

    //Zápis do buffera//
    IF Buffer_17.ZapisHodnotu THEN
        Buffer_17.Pole[Buffer_17.Index]:= Buffer_17.Hodnota;
        IF Buffer_17.Index < 100 THEN
            Buffer_17.Index:= Buffer_17.Index + 1;
        ELSE
            Buffer_17.Index:= 0;
        END_IF
        Buffer_17.ZapisHodnotu:= FALSE;
    END_IF

	//*********************************************Buffer 18****************************************************//
	//Resetovanie//
	IF Buffer_18.ResetBufferu THEN
		brsmemset(ADR(Buffer_18.Pole),0,SIZEOF(Buffer_18.Pole));
		Buffer_18.Index:= 0;
		Buffer_18.ResetBufferu:= FALSE;
	END_IF

	//Zápis do buffera//
	IF Buffer_18.ZapisHodnotu THEN
		Buffer_18.Pole[Buffer_18.Index]:= Buffer_18.Hodnota;
		IF Buffer_18.Index < 100 THEN
			Buffer_18.Index:= Buffer_18.Index + 1;
		ELSE
			Buffer_18.Index:= 0;
		END_IF
		Buffer_18.ZapisHodnotu:= FALSE;
	END_IF

	//*********************************************Buffer 19****************************************************//
	//Resetovanie//
	IF Buffer_19.ResetBufferu THEN
		brsmemset(ADR(Buffer_19.Pole),0,SIZEOF(Buffer_19.Pole));
		Buffer_19.Index:= 0;
		Buffer_19.ResetBufferu:= FALSE;
	END_IF

	//Zápis do buffera//
	IF Buffer_19.ZapisHodnotu THEN
		Buffer_19.Pole[Buffer_19.Index]:= Buffer_19.Hodnota;
		IF Buffer_19.Index < 100 THEN
			Buffer_19.Index:= Buffer_19.Index + 1;
		ELSE
			Buffer_19.Index:= 0;
		END_IF
		Buffer_19.ZapisHodnotu:= FALSE;
	END_IF

	//*********************************************Buffer 20****************************************************//
	//Resetovanie//
	IF Buffer_20.ResetBufferu THEN
		brsmemset(ADR(Buffer_20.Pole),0,SIZEOF(Buffer_20.Pole));
		Buffer_20.Index:= 0;
		Buffer_20.ResetBufferu:= FALSE;
	END_IF

	//Zápis do buffera//
	IF Buffer_20.ZapisHodnotu THEN
		Buffer_20.Pole[Buffer_20.Index]:= Buffer_20.Hodnota;
		IF Buffer_20.Index < 100 THEN
			Buffer_20.Index:= Buffer_20.Index + 1;
		ELSE
			Buffer_20.Index:= 0;
		END_IF
		Buffer_20.ZapisHodnotu:= FALSE;
	END_IF

END_PROGRAM

PROGRAM _EXIT
	(* Insert code here *)

END_PROGRAM
```

### Program Logical/TracebilitySystem/P1_Vytah_ST1 (IEC)
